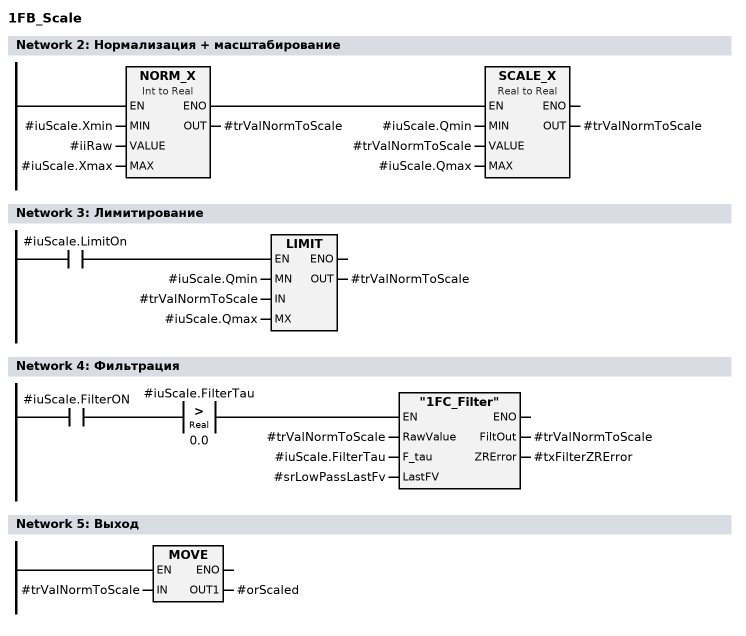
   RUNG wire#powerrail
      { S7_Templates := "[SrcType := Int, DestType := Real]" } Normalize(min := #iuScale.Xmin, value := #iiRaw, max := #iuScale.Xmax, out => #trValNormToScale)
      { S7_Templates := "[SrcType := Real, DestType := Real]" } Scale(min := #iuScale.Qmin, value := #trValNormToScale, max := #iuScale.Qmax, out => #trValNormToScale)
   END_RUNG
   // the same network as SCL:
   #trValNormToScale := NORM_X(MIN := #iuScale.Xmin, VALUE := #iiRaw, MAX := #iuScale.Xmax);
   #trValNormToScale := SCALE_X(MIN := #iuScale.Qmin, VALUE := #trValNormToScale, MAX := #iuScale.Qmax);
END_REGION

REGION Network 3: Лимитирование
   IF #iuScale.LimitOn THEN
       #trValNormToScale := LIMIT(MN := #iuScale.Qmin, IN := #trValNormToScale, MX := #iuScale.Qmax);
   END_IF;
END_REGION

REGION Network 4: Фильтрация
   RUNG wire#powerrail
      Contact( #iuScale.FilterON )
      { S7_Templates := "SrcType := Real" } GT_Contact(in1 := #iuScale.FilterTau, in2 := 0.0)
      "1FC_Filter"(RawValue := #trValNormToScale, F_tau := #iuScale.FilterTau, LastFV := #srLowPassLastFv, FiltOut => #trValNormToScale, ZRError => #txFilterZRError)
   END_RUNG
   // the same network as SCL:
   IF #iuScale.FilterON AND (#iuScale.FilterTau > 0.0) THEN
       "1FC_Filter"(RawValue := #trValNormToScale,
                    F_tau := #iuScale.FilterTau,
                    LastFV := #srLowPassLastFv,
                    FiltOut => #trValNormToScale,
                    ZRError => #txFilterZRError);
   END_IF;
END_REGION

REGION Network 5: Выход
   RUNG wire#powerrail
      Move(in := #trValNormToScale, out1 => #orScaled)
   END_RUNG
   // the same network as SCL:
   #orScaled := #trValNormToScale;
END_REGION
END_FUNCTION_BLOCK

FUNCTION_BLOCK "1FB_ScaleRTD"   // FB131, LAD
TITLE = Физ.значение аналогового входа термометра
{ S7_Optimized_Access := 'TRUE' }
VERSION : 0.1
// Преорбазование аналогового входа термрметра сопротивления в физ.значение согласно шкалы
   VAR_INPUT
      iiRaw : Int;   // Входной сигнал
      iuScale : "uScale";
   END_VAR
   VAR_OUTPUT
      orScaled : Real;   // Выходное отмасштабированное значение
   END_VAR
   VAR
      srLowPassLastFv : Real;   // Выходное значение для следующего цикла расчета
   END_VAR
   VAR_TEMP
      trValNormToScale : Real;   // Временная переменная
      txFilterZRError : Bool;   // Ошибка, если t = 0,0s
   END_VAR
BEGIN

REGION Network 2 (SCL): Временная переменная
   #trValNormToScale := INT_TO_REAL(#iiRaw);
END_REGION

REGION Network 3: Нормализация + масштабирование
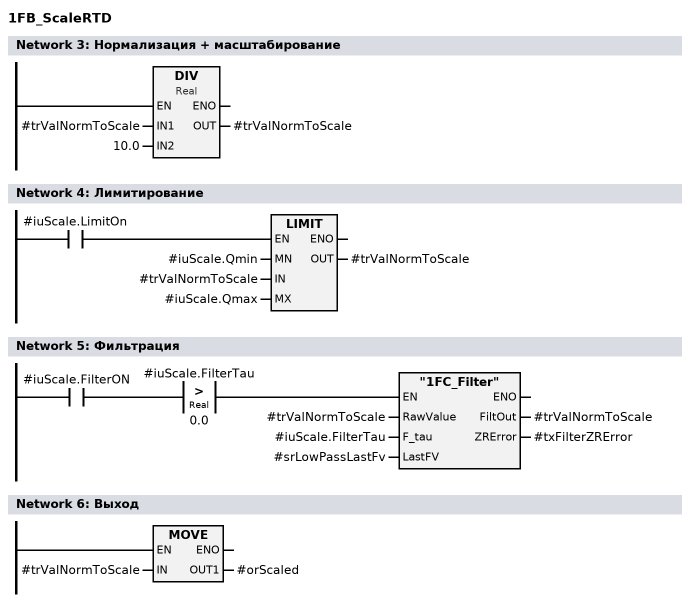
   RUNG wire#powerrail
      { S7_Templates := "SrcType := Real" } Div(in1 := #trValNormToScale, in2 := 10.0, out => #trValNormToScale)
   END_RUNG
   // the same network as SCL:
   #trValNormToScale := #trValNormToScale / 10.0;
END_REGION

REGION Network 4: Лимитирование
   IF #iuScale.LimitOn THEN
       #trValNormToScale := LIMIT(MN := #iuScale.Qmin, IN := #trValNormToScale, MX := #iuScale.Qmax);
   END_IF;
END_REGION

REGION Network 5: Фильтрация
   RUNG wire#powerrail
      Contact( #iuScale.FilterON )
      { S7_Templates := "SrcType := Real" } GT_Contact(in1 := #iuScale.FilterTau, in2 := 0.0)
      "1FC_Filter"(RawValue := #trValNormToScale, F_tau := #iuScale.FilterTau, LastFV := #srLowPassLastFv, FiltOut => #trValNormToScale, ZRError => #txFilterZRError)
   END_RUNG
   // the same network as SCL:
   IF #iuScale.FilterON AND (#iuScale.FilterTau > 0.0) THEN
       "1FC_Filter"(RawValue := #trValNormToScale,
                    F_tau := #iuScale.FilterTau,
                    LastFV := #srLowPassLastFv,
                    FiltOut => #trValNormToScale,
                    ZRError => #txFilterZRError);
   END_IF;
END_REGION

REGION Network 6: Выход
   RUNG wire#powerrail
      Move(in := #trValNormToScale, out1 => #orScaled)
   END_RUNG
   // the same network as SCL:
   #orScaled := #trValNormToScale;
END_REGION
END_FUNCTION_BLOCK

FUNCTION "1FC_Limit" : Void   // FC104, LAD
TITLE = Ааварийные и предупредительные границы
{ S7_Optimized_Access := 'TRUE' }
VERSION : 0.1
// Функция проверки аварийных и предупредительных границ аналогового сигнала, чтобы
// НШ <= НАГ <= НПГ <= ВПГ <= ВАГ <= КШ 
// НШ - начало шкалы
// НАГ - нижняя аварийная граница
// НПГ - нижняя предупредительная граница и тд
   VAR_INPUT
      inAI : "uScale";
   END_VAR
   VAR_IN_OUT
      ioWarning : "uWrnngAlarm";
      ioAlarm : "uWrnngAlarm";
   END_VAR
BEGIN

REGION Network 2: Если НАГ > НПГ и ниже если НАГ < НШ
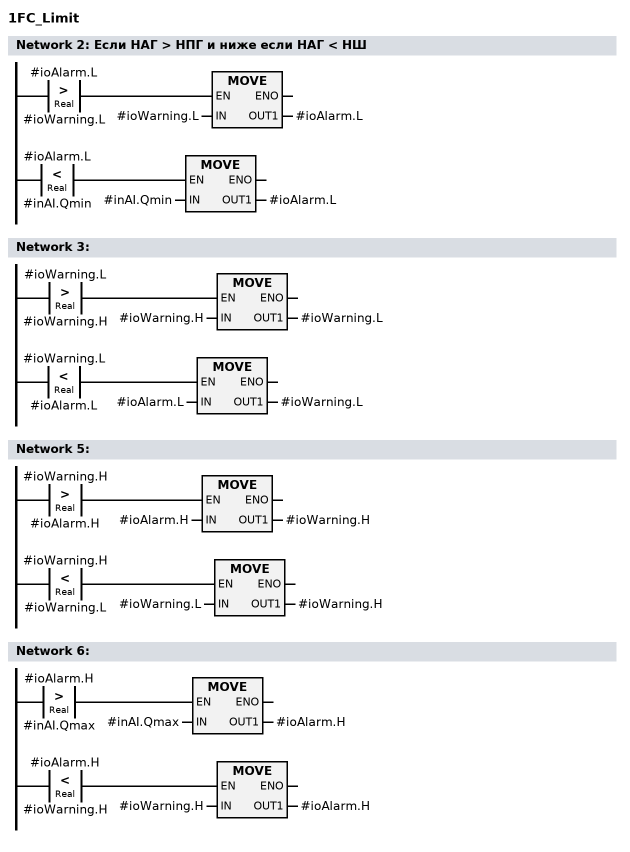
   RUNG wire#powerrail
      { S7_Templates := "SrcType := Real" } GT_Contact(in1 := #ioAlarm.L, in2 := #ioWarning.L)
      Move(in := #ioWarning.L, out1 => #ioAlarm.L)
   END_RUNG
   RUNG wire#powerrail
      { S7_Templates := "SrcType := Real" } LT_Contact(in1 := #ioAlarm.L, in2 := #inAI.Qmin)
      Move(in := #inAI.Qmin, out1 => #ioAlarm.L)
   END_RUNG
   // the same network as SCL:
   IF #ioAlarm.L > #ioWarning.L THEN #ioAlarm.L := #ioWarning.L; END_IF;
   IF #ioAlarm.L < #inAI.Qmin THEN #ioAlarm.L := #inAI.Qmin; END_IF;
END_REGION

REGION Network 3
   RUNG wire#powerrail
      { S7_Templates := "SrcType := Real" } GT_Contact(in1 := #ioWarning.L, in2 := #ioWarning.H)
      Move(in := #ioWarning.H, out1 => #ioWarning.L)
   END_RUNG
   RUNG wire#powerrail
      { S7_Templates := "SrcType := Real" } LT_Contact(in1 := #ioWarning.L, in2 := #ioAlarm.L)
      Move(in := #ioAlarm.L, out1 => #ioWarning.L)
   END_RUNG
   // the same network as SCL:
   IF #ioWarning.L > #ioWarning.H THEN #ioWarning.L := #ioWarning.H; END_IF;
   IF #ioWarning.L < #ioAlarm.L THEN #ioWarning.L := #ioAlarm.L; END_IF;
END_REGION

REGION Network 5
   RUNG wire#powerrail
      { S7_Templates := "SrcType := Real" } GT_Contact(in1 := #ioWarning.H, in2 := #ioAlarm.H)
      Move(in := #ioAlarm.H, out1 => #ioWarning.H)
   END_RUNG
   RUNG wire#powerrail
      { S7_Templates := "SrcType := Real" } LT_Contact(in1 := #ioWarning.H, in2 := #ioWarning.L)
      Move(in := #ioWarning.L, out1 => #ioWarning.H)
   END_RUNG
   // the same network as SCL:
   IF #ioWarning.H > #ioAlarm.H THEN #ioWarning.H := #ioAlarm.H; END_IF;
   IF #ioWarning.H < #ioWarning.L THEN #ioWarning.H := #ioWarning.L; END_IF;
END_REGION

REGION Network 6
   RUNG wire#powerrail
      { S7_Templates := "SrcType := Real" } GT_Contact(in1 := #ioAlarm.H, in2 := #inAI.Qmax)
      Move(in := #inAI.Qmax, out1 => #ioAlarm.H)
   END_RUNG
   RUNG wire#powerrail
      { S7_Templates := "SrcType := Real" } LT_Contact(in1 := #ioAlarm.H, in2 := #ioWarning.H)
      Move(in := #ioWarning.H, out1 => #ioAlarm.H)
   END_RUNG
   // the same network as SCL:
   IF #ioAlarm.H > #inAI.Qmax THEN #ioAlarm.H := #inAI.Qmax; END_IF;
   IF #ioAlarm.H < #ioWarning.H THEN #ioAlarm.H := #ioWarning.H; END_IF;
END_REGION
END_FUNCTION

FUNCTION "1FC_FlowNorm" : Void   // FC105, LAD
TITLE = Нормальный расход
{ S7_Optimized_Access := 'TRUE' }
VERSION : 0.1
// Нормализация расхода газа (не для расхода жидкости)
   VAR_INPUT
      inScaled : Real;
   END_VAR
   VAR_OUTPUT
      outScaledNorm : Real;
   END_VAR
BEGIN

REGION Network 2 (SCL)
   #outScaledNorm := #inScaled;
END_REGION
END_FUNCTION

FUNCTION "1FC_Filter" : Void   // FC106, SCL
TITLE = Фильтр низких частот
{ S7_Optimized_Access := 'TRUE' }
VERSION : 0.1
// Функция фильтрации аналогового входа
   VAR_INPUT
      RawValue : Real;   // Incoming unfiltered value
      F_tau : Real;   // Time interval (in seconds) for filter period
   END_VAR
   VAR_OUTPUT
      FiltOut : Real;   // Filtered output value
      ZRError : Bool;   // Error flag if F_tau is set to zero (invalid rate)
   END_VAR
   VAR_IN_OUT
      LastFV : Real;   // Static variable holds value of FiltOut from previous execution cycle.
   END_VAR
   VAR_TEMP
      ExpRate : Real;   // Equals exp(-0.1 / F_tau)
   END_VAR
BEGIN

   (* ============================================================================= *)
   (* PURPOSE : To filter a value by applying a first-order exponential filter      *)
   (*           with a user-selectable time period, F-tau. The filter is calculated *)
   (*           using the following formula -                                       *)
   (*                                                                               *)
   (*                                 Rate                    Rate                  *)
   (*           FiltOut := FiltOut * e     + RawValue * (1 - e     )                *)
   (*                                                                               *)
   (*           where Rate := (-0.1 / F_tau )                                       *)
   (*                                                                               *)
   (*           The Function Block is intended to be triggered every 100mS (hence   *)
   (*           the 0.1 in the formula) from cyclic interrupt Organization Block    *)
   (*           OB35. If a different resolution is required, use a different OB as  *)
   (*           the trigger, and adjust the formula to reflect this.                *)                                                                    
   (*                                                                               *)
   (* ============================================================================= *)


   IF #F_tau = 0.0 THEN                                        // If the filter period is set to zero ...
       #ZRError := true;                                     // .. . set the Zero Rate Error bit true
   ELSE
       #ZRError := false;                                       // Error bit reset to false
       #ExpRate := EXP(-0.1 / #F_tau);
       #FiltOut := #LastFV * #ExpRate + (#RawValue * (1 - #ExpRate)); // Calculate new output
       #LastFV := #FiltOut;                                       // Store output value for next cycle of calculation
   END_IF;
END_FUNCTION

FUNCTION "AI_Scaling" : Void   // FC131, LAD
TITLE = Физ.значение для всех аналог.сигналов
{ S7_Optimized_Access := 'TRUE' }
VERSION : 0.1
// Расчет физических значений всех аналоговых сигналов
   VAR_TEMP
      rTemp : Real;
   END_VAR
   VAR_TEMP   // added for the SCL form of the ladder/FBD networks
      _w1 : Bool;
   END_VAR
BEGIN

REGION Network 1: Разрежение на газоходе перед циклоном PIT201a
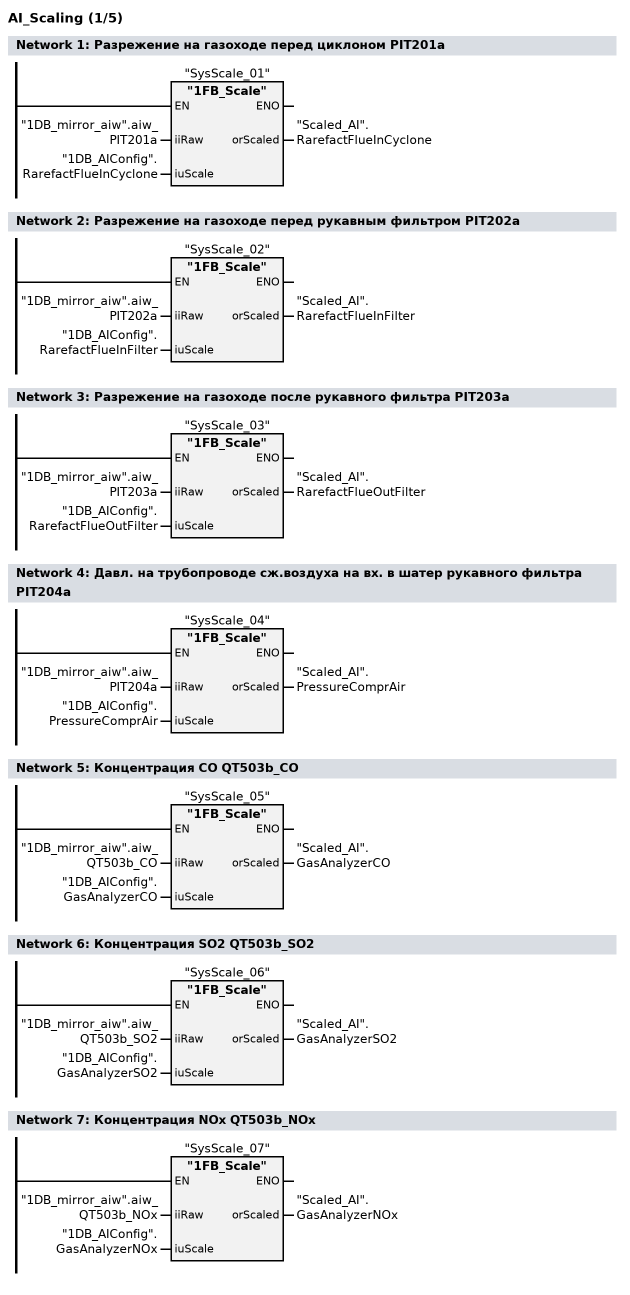
   RUNG wire#powerrail
      "SysScale_01"(iiRaw := "1DB_mirror_aiw".aiw_PIT201a, iuScale := "1DB_AIConfig".RarefactFlueInCyclone, orScaled => "Scaled_AI".RarefactFlueInCyclone)
   END_RUNG
   // the same network as SCL:
   "SysScale_01"(iiRaw := "1DB_mirror_aiw".aiw_PIT201a,   // "1FB_Scale"
                 iuScale := "1DB_AIConfig".RarefactFlueInCyclone,
                 orScaled => "Scaled_AI".RarefactFlueInCyclone);
END_REGION

REGION Network 2: Разрежение на газоходе перед рукавным фильтром PIT202a
   RUNG wire#powerrail
      "SysScale_02"(iiRaw := "1DB_mirror_aiw".aiw_PIT202a, iuScale := "1DB_AIConfig".RarefactFlueInFilter, orScaled => "Scaled_AI".RarefactFlueInFilter)
   END_RUNG
   // the same network as SCL:
   "SysScale_02"(iiRaw := "1DB_mirror_aiw".aiw_PIT202a,   // "1FB_Scale"
                 iuScale := "1DB_AIConfig".RarefactFlueInFilter,
                 orScaled => "Scaled_AI".RarefactFlueInFilter);
END_REGION

REGION Network 3: Разрежение на газоходе после рукавного фильтра PIT203a
   RUNG wire#powerrail
      "SysScale_03"(iiRaw := "1DB_mirror_aiw".aiw_PIT203a, iuScale := "1DB_AIConfig".RarefactFlueOutFilter, orScaled => "Scaled_AI".RarefactFlueOutFilter)
   END_RUNG
   // the same network as SCL:
   "SysScale_03"(iiRaw := "1DB_mirror_aiw".aiw_PIT203a,   // "1FB_Scale"
                 iuScale := "1DB_AIConfig".RarefactFlueOutFilter,
                 orScaled => "Scaled_AI".RarefactFlueOutFilter);
END_REGION

REGION Network 4: Давл. на трубопроводе сж.воздуха на вх. в шатер рукавного фильтра PIT204a
   RUNG wire#powerrail
      "SysScale_04"(iiRaw := "1DB_mirror_aiw".aiw_PIT204a, iuScale := "1DB_AIConfig".PressureComprAir, orScaled => "Scaled_AI".PressureComprAir)
   END_RUNG
   // the same network as SCL:
   "SysScale_04"(iiRaw := "1DB_mirror_aiw".aiw_PIT204a,   // "1FB_Scale"
                 iuScale := "1DB_AIConfig".PressureComprAir,
                 orScaled => "Scaled_AI".PressureComprAir);
END_REGION

REGION Network 5: Концентрация CO QT503b_CO
   RUNG wire#powerrail
      "SysScale_05"(iiRaw := "1DB_mirror_aiw".aiw_QT503b_CO, iuScale := "1DB_AIConfig".GasAnalyzerCO, orScaled => "Scaled_AI".GasAnalyzerCO)
   END_RUNG
   // the same network as SCL:
   "SysScale_05"(iiRaw := "1DB_mirror_aiw".aiw_QT503b_CO,   // "1FB_Scale"
                 iuScale := "1DB_AIConfig".GasAnalyzerCO,
                 orScaled => "Scaled_AI".GasAnalyzerCO);
END_REGION

REGION Network 6: Концентрация SO2 QT503b_SO2
   RUNG wire#powerrail
      "SysScale_06"(iiRaw := "1DB_mirror_aiw".aiw_QT503b_SO2, iuScale := "1DB_AIConfig".GasAnalyzerSO2, orScaled => "Scaled_AI".GasAnalyzerSO2)
   END_RUNG
   // the same network as SCL:
   "SysScale_06"(iiRaw := "1DB_mirror_aiw".aiw_QT503b_SO2,   // "1FB_Scale"
                 iuScale := "1DB_AIConfig".GasAnalyzerSO2,
                 orScaled => "Scaled_AI".GasAnalyzerSO2);
END_REGION

REGION Network 7: Концентрация NOx QT503b_NOx
   RUNG wire#powerrail
      "SysScale_07"(iiRaw := "1DB_mirror_aiw".aiw_QT503b_NOx, iuScale := "1DB_AIConfig".GasAnalyzerNOx, orScaled => "Scaled_AI".GasAnalyzerNOx)
   END_RUNG
   // the same network as SCL:
   "SysScale_07"(iiRaw := "1DB_mirror_aiw".aiw_QT503b_NOx,   // "1FB_Scale"
                 iuScale := "1DB_AIConfig".GasAnalyzerNOx,
                 orScaled => "Scaled_AI".GasAnalyzerNOx);
END_REGION

REGION Network 8: Концентрация CO2 QT503b_CO2
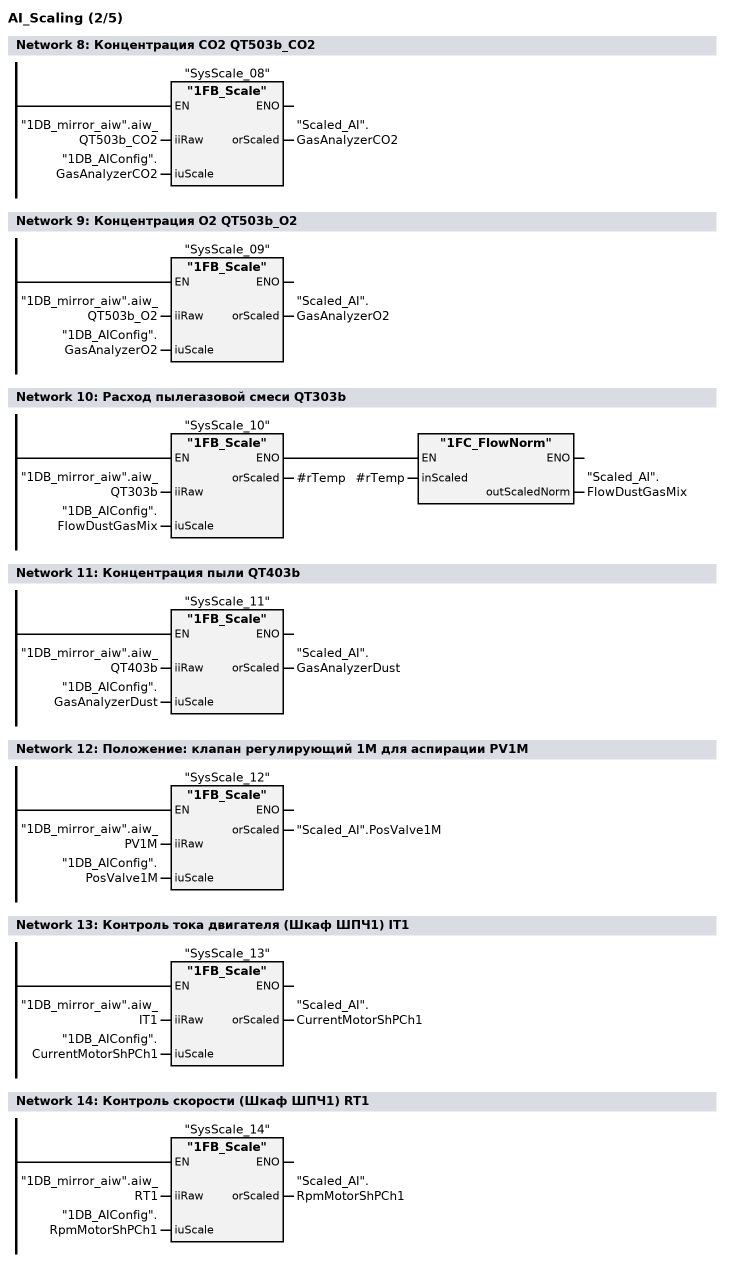
   RUNG wire#powerrail
      "SysScale_08"(iiRaw := "1DB_mirror_aiw".aiw_QT503b_CO2, iuScale := "1DB_AIConfig".GasAnalyzerCO2, orScaled => "Scaled_AI".GasAnalyzerCO2)
   END_RUNG
   // the same network as SCL:
   "SysScale_08"(iiRaw := "1DB_mirror_aiw".aiw_QT503b_CO2,   // "1FB_Scale"
                 iuScale := "1DB_AIConfig".GasAnalyzerCO2,
                 orScaled => "Scaled_AI".GasAnalyzerCO2);
END_REGION

REGION Network 9: Концентрация O2 QT503b_O2
   RUNG wire#powerrail
      "SysScale_09"(iiRaw := "1DB_mirror_aiw".aiw_QT503b_O2, iuScale := "1DB_AIConfig".GasAnalyzerO2, orScaled => "Scaled_AI".GasAnalyzerO2)
   END_RUNG
   // the same network as SCL:
   "SysScale_09"(iiRaw := "1DB_mirror_aiw".aiw_QT503b_O2,   // "1FB_Scale"
                 iuScale := "1DB_AIConfig".GasAnalyzerO2,
                 orScaled => "Scaled_AI".GasAnalyzerO2);
END_REGION

REGION Network 10: Расход пылегазовой смеси QT303b
   RUNG wire#powerrail
      "SysScale_10"(iiRaw := "1DB_mirror_aiw".aiw_QT303b, iuScale := "1DB_AIConfig".FlowDustGasMix, orScaled => #rTemp)
      "1FC_FlowNorm"(inScaled := #rTemp, outScaledNorm => "Scaled_AI".FlowDustGasMix)
   END_RUNG
   // the same network as SCL:
   "SysScale_10"(iiRaw := "1DB_mirror_aiw".aiw_QT303b,   // "1FB_Scale"
                 iuScale := "1DB_AIConfig".FlowDustGasMix,
                 orScaled => #rTemp,
                 ENO => #_w1);
   IF #_w1 THEN "1FC_FlowNorm"(inScaled := #rTemp, outScaledNorm => "Scaled_AI".FlowDustGasMix); END_IF;
END_REGION

REGION Network 11: Концентрация пыли QT403b
   RUNG wire#powerrail
      "SysScale_11"(iiRaw := "1DB_mirror_aiw".aiw_QT403b, iuScale := "1DB_AIConfig".GasAnalyzerDust, orScaled => "Scaled_AI".GasAnalyzerDust)
   END_RUNG
   // the same network as SCL:
   "SysScale_11"(iiRaw := "1DB_mirror_aiw".aiw_QT403b,   // "1FB_Scale"
                 iuScale := "1DB_AIConfig".GasAnalyzerDust,
                 orScaled => "Scaled_AI".GasAnalyzerDust);
END_REGION

REGION Network 12: Положение: клапан регулирующий 1M для аспирации PV1M
   RUNG wire#powerrail
      "SysScale_12"(iiRaw := "1DB_mirror_aiw".aiw_PV1M, iuScale := "1DB_AIConfig".PosValve1M, orScaled => "Scaled_AI".PosValve1M)
   END_RUNG
   // the same network as SCL:
   "SysScale_12"(iiRaw := "1DB_mirror_aiw".aiw_PV1M,   // "1FB_Scale"
                 iuScale := "1DB_AIConfig".PosValve1M,
                 orScaled => "Scaled_AI".PosValve1M);
END_REGION

REGION Network 13: Контроль тока двигателя (Шкаф ШПЧ1) IT1
   RUNG wire#powerrail
      "SysScale_13"(iiRaw := "1DB_mirror_aiw".aiw_IT1, iuScale := "1DB_AIConfig".CurrentMotorShPCh1, orScaled => "Scaled_AI".CurrentMotorShPCh1)
   END_RUNG
   // the same network as SCL:
   "SysScale_13"(iiRaw := "1DB_mirror_aiw".aiw_IT1,   // "1FB_Scale"
                 iuScale := "1DB_AIConfig".CurrentMotorShPCh1,
                 orScaled => "Scaled_AI".CurrentMotorShPCh1);
END_REGION

REGION Network 14: Контроль скорости (Шкаф ШПЧ1) RT1
   RUNG wire#powerrail
      "SysScale_14"(iiRaw := "1DB_mirror_aiw".aiw_RT1, iuScale := "1DB_AIConfig".RpmMotorShPCh1, orScaled => "Scaled_AI".RpmMotorShPCh1)
   END_RUNG
   // the same network as SCL:
   "SysScale_14"(iiRaw := "1DB_mirror_aiw".aiw_RT1,   // "1FB_Scale"
                 iuScale := "1DB_AIConfig".RpmMotorShPCh1,
                 orScaled => "Scaled_AI".RpmMotorShPCh1);
END_REGION

REGION Network 15: 2 резервных места
END_REGION

REGION Network 16: 2 резервных места
END_REGION

REGION Network 17: Дымосос 1. Вибрация переднего подшипника вентилятора X-направления VE801a
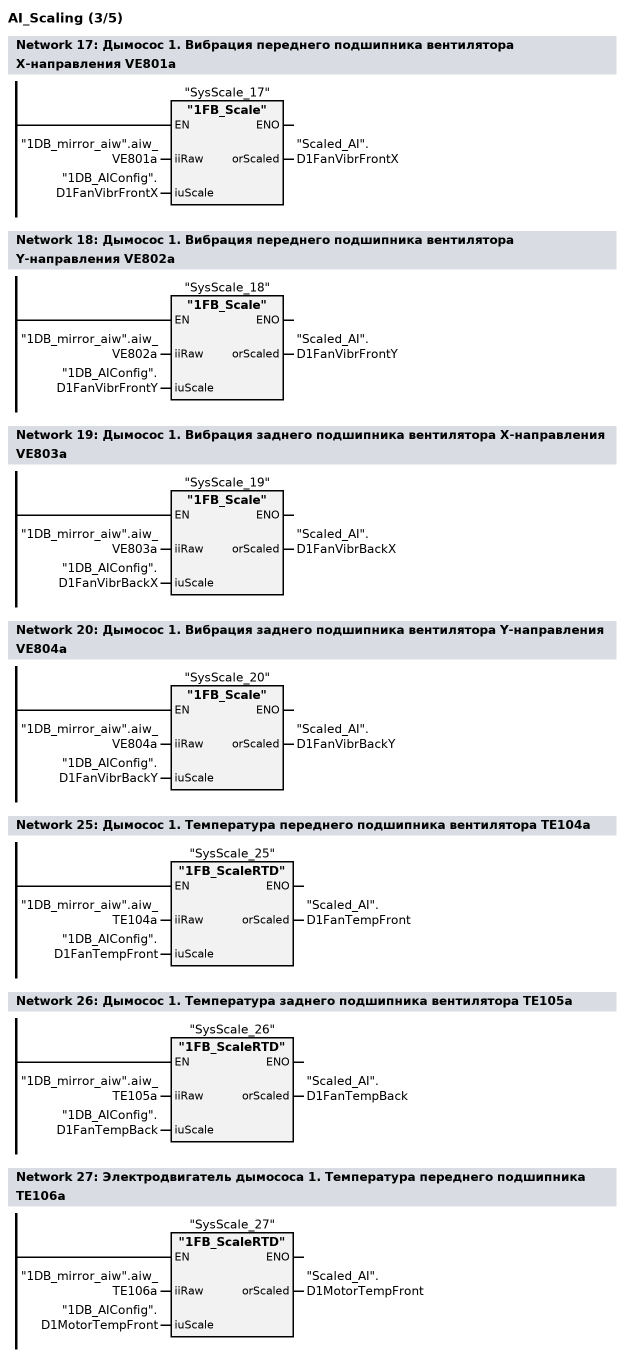
   RUNG wire#powerrail
      "SysScale_17"(iiRaw := "1DB_mirror_aiw".aiw_VE801a, iuScale := "1DB_AIConfig".D1FanVibrFrontX, orScaled => "Scaled_AI".D1FanVibrFrontX)
   END_RUNG
   // the same network as SCL:
   "SysScale_17"(iiRaw := "1DB_mirror_aiw".aiw_VE801a,   // "1FB_Scale"
                 iuScale := "1DB_AIConfig".D1FanVibrFrontX,
                 orScaled => "Scaled_AI".D1FanVibrFrontX);
END_REGION

REGION Network 18: Дымосос 1. Вибрация переднего подшипника вентилятора Y-направления VE802a
   RUNG wire#powerrail
      "SysScale_18"(iiRaw := "1DB_mirror_aiw".aiw_VE802a, iuScale := "1DB_AIConfig".D1FanVibrFrontY, orScaled => "Scaled_AI".D1FanVibrFrontY)
   END_RUNG
   // the same network as SCL:
   "SysScale_18"(iiRaw := "1DB_mirror_aiw".aiw_VE802a,   // "1FB_Scale"
                 iuScale := "1DB_AIConfig".D1FanVibrFrontY,
                 orScaled => "Scaled_AI".D1FanVibrFrontY);
END_REGION

REGION Network 19: Дымосос 1. Вибрация заднего подшипника вентилятора X-направления VE803a
   RUNG wire#powerrail
      "SysScale_19"(iiRaw := "1DB_mirror_aiw".aiw_VE803a, iuScale := "1DB_AIConfig".D1FanVibrBackX, orScaled => "Scaled_AI".D1FanVibrBackX)
   END_RUNG
   // the same network as SCL:
   "SysScale_19"(iiRaw := "1DB_mirror_aiw".aiw_VE803a,   // "1FB_Scale"
                 iuScale := "1DB_AIConfig".D1FanVibrBackX,
                 orScaled => "Scaled_AI".D1FanVibrBackX);
END_REGION

REGION Network 20: Дымосос 1. Вибрация заднего подшипника вентилятора Y-направления VE804a
   RUNG wire#powerrail
      "SysScale_20"(iiRaw := "1DB_mirror_aiw".aiw_VE804a, iuScale := "1DB_AIConfig".D1FanVibrBackY, orScaled => "Scaled_AI".D1FanVibrBackY)
   END_RUNG
   // the same network as SCL:
   "SysScale_20"(iiRaw := "1DB_mirror_aiw".aiw_VE804a,   // "1FB_Scale"
                 iuScale := "1DB_AIConfig".D1FanVibrBackY,
                 orScaled => "Scaled_AI".D1FanVibrBackY);
END_REGION

REGION Network 21: 4 резервных места
END_REGION

REGION Network 22: 4 резервных места
END_REGION

REGION Network 23: 4 резервных места
END_REGION

REGION Network 24: 4 резервных места
END_REGION

REGION Network 25: Дымосос 1. Температура переднего подшипника вентилятора TE104a
   RUNG wire#powerrail
      "SysScale_25"(iiRaw := "1DB_mirror_aiw".aiw_TE104a, iuScale := "1DB_AIConfig".D1FanTempFront, orScaled => "Scaled_AI".D1FanTempFront)
   END_RUNG
   // the same network as SCL:
   "SysScale_25"(iiRaw := "1DB_mirror_aiw".aiw_TE104a,   // "1FB_ScaleRTD"
                 iuScale := "1DB_AIConfig".D1FanTempFront,
                 orScaled => "Scaled_AI".D1FanTempFront);
END_REGION

REGION Network 26: Дымосос 1. Температура заднего подшипника вентилятора TE105a
   RUNG wire#powerrail
      "SysScale_26"(iiRaw := "1DB_mirror_aiw".aiw_TE105a, iuScale := "1DB_AIConfig".D1FanTempBack, orScaled => "Scaled_AI".D1FanTempBack)
   END_RUNG
   // the same network as SCL:
   "SysScale_26"(iiRaw := "1DB_mirror_aiw".aiw_TE105a,   // "1FB_ScaleRTD"
                 iuScale := "1DB_AIConfig".D1FanTempBack,
                 orScaled => "Scaled_AI".D1FanTempBack);
END_REGION

REGION Network 27: Электродвигатель дымососа 1. Температура переднего подшипника TE106a
   RUNG wire#powerrail
      "SysScale_27"(iiRaw := "1DB_mirror_aiw".aiw_TE106a, iuScale := "1DB_AIConfig".D1MotorTempFront, orScaled => "Scaled_AI".D1MotorTempFront)
   END_RUNG
   // the same network as SCL:
   "SysScale_27"(iiRaw := "1DB_mirror_aiw".aiw_TE106a,   // "1FB_ScaleRTD"
                 iuScale := "1DB_AIConfig".D1MotorTempFront,
                 orScaled => "Scaled_AI".D1MotorTempFront);
END_REGION

REGION Network 28: Электродвигатель дымососа 1. Температура заднего подшипника TE107a
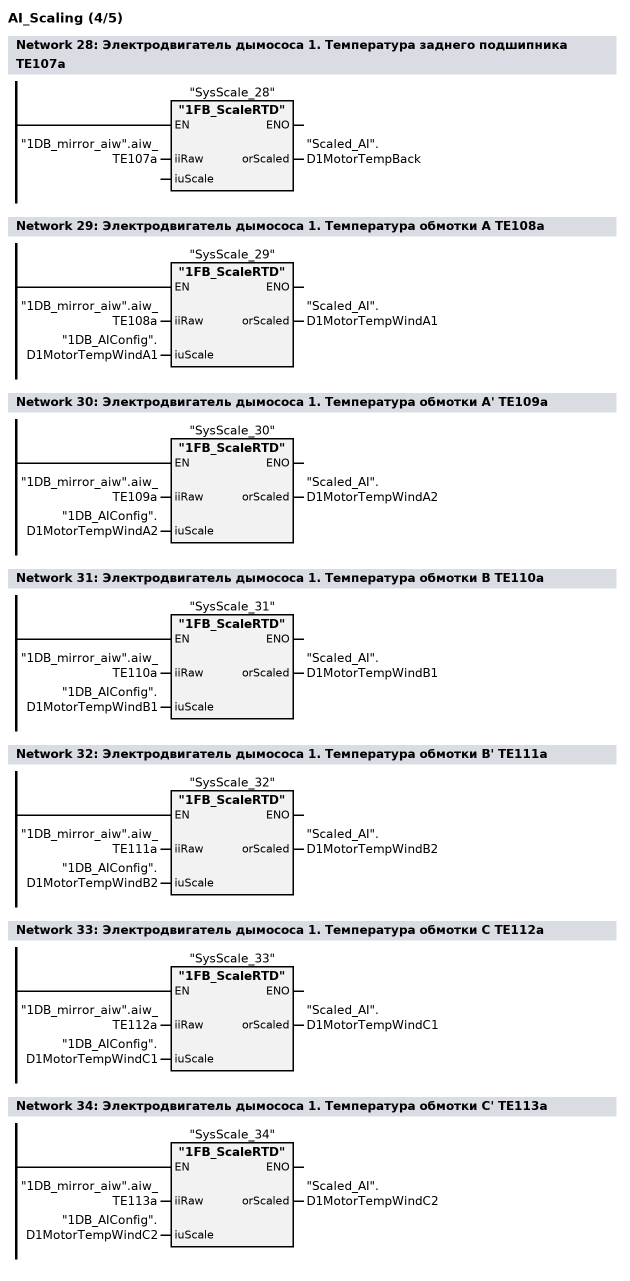
   RUNG wire#powerrail
      "SysScale_28"(iiRaw := "1DB_mirror_aiw".aiw_TE107a, iuScale :=, orScaled => "Scaled_AI".D1MotorTempBack)
   END_RUNG
   // the same network as SCL:
   "SysScale_28"(iiRaw := "1DB_mirror_aiw".aiw_TE107a, orScaled => "Scaled_AI".D1MotorTempBack);   // "1FB_ScaleRTD"
END_REGION

REGION Network 29: Электродвигатель дымососа 1. Температура обмотки А TE108a
   RUNG wire#powerrail
      "SysScale_29"(iiRaw := "1DB_mirror_aiw".aiw_TE108a, iuScale := "1DB_AIConfig".D1MotorTempWindA1, orScaled => "Scaled_AI".D1MotorTempWindA1)
   END_RUNG
   // the same network as SCL:
   "SysScale_29"(iiRaw := "1DB_mirror_aiw".aiw_TE108a,   // "1FB_ScaleRTD"
                 iuScale := "1DB_AIConfig".D1MotorTempWindA1,
                 orScaled => "Scaled_AI".D1MotorTempWindA1);
END_REGION

REGION Network 30: Электродвигатель дымососа 1. Температура обмотки А' TE109a
   RUNG wire#powerrail
      "SysScale_30"(iiRaw := "1DB_mirror_aiw".aiw_TE109a, iuScale := "1DB_AIConfig".D1MotorTempWindA2, orScaled => "Scaled_AI".D1MotorTempWindA2)
   END_RUNG
   // the same network as SCL:
   "SysScale_30"(iiRaw := "1DB_mirror_aiw".aiw_TE109a,   // "1FB_ScaleRTD"
                 iuScale := "1DB_AIConfig".D1MotorTempWindA2,
                 orScaled => "Scaled_AI".D1MotorTempWindA2);
END_REGION

REGION Network 31: Электродвигатель дымососа 1. Температура обмотки B TE110a
   RUNG wire#powerrail
      "SysScale_31"(iiRaw := "1DB_mirror_aiw".aiw_TE110a, iuScale := "1DB_AIConfig".D1MotorTempWindB1, orScaled => "Scaled_AI".D1MotorTempWindB1)
   END_RUNG
   // the same network as SCL:
   "SysScale_31"(iiRaw := "1DB_mirror_aiw".aiw_TE110a,   // "1FB_ScaleRTD"
                 iuScale := "1DB_AIConfig".D1MotorTempWindB1,
                 orScaled => "Scaled_AI".D1MotorTempWindB1);
END_REGION

REGION Network 32: Электродвигатель дымососа 1. Температура обмотки B' TE111a
   RUNG wire#powerrail
      "SysScale_32"(iiRaw := "1DB_mirror_aiw".aiw_TE111a, iuScale := "1DB_AIConfig".D1MotorTempWindB2, orScaled => "Scaled_AI".D1MotorTempWindB2)
   END_RUNG
   // the same network as SCL:
   "SysScale_32"(iiRaw := "1DB_mirror_aiw".aiw_TE111a,   // "1FB_ScaleRTD"
                 iuScale := "1DB_AIConfig".D1MotorTempWindB2,
                 orScaled => "Scaled_AI".D1MotorTempWindB2);
END_REGION

REGION Network 33: Электродвигатель дымососа 1. Температура обмотки C TE112a
   RUNG wire#powerrail
      "SysScale_33"(iiRaw := "1DB_mirror_aiw".aiw_TE112a, iuScale := "1DB_AIConfig".D1MotorTempWindC1, orScaled => "Scaled_AI".D1MotorTempWindC1)
   END_RUNG
   // the same network as SCL:
   "SysScale_33"(iiRaw := "1DB_mirror_aiw".aiw_TE112a,   // "1FB_ScaleRTD"
                 iuScale := "1DB_AIConfig".D1MotorTempWindC1,
                 orScaled => "Scaled_AI".D1MotorTempWindC1);
END_REGION

REGION Network 34: Электродвигатель дымососа 1. Температура обмотки C' TE113a
   RUNG wire#powerrail
      "SysScale_34"(iiRaw := "1DB_mirror_aiw".aiw_TE113a, iuScale := "1DB_AIConfig".D1MotorTempWindC2, orScaled => "Scaled_AI".D1MotorTempWindC2)
   END_RUNG
   // the same network as SCL:
   "SysScale_34"(iiRaw := "1DB_mirror_aiw".aiw_TE113a,   // "1FB_ScaleRTD"
                 iuScale := "1DB_AIConfig".D1MotorTempWindC2,
                 orScaled => "Scaled_AI".D1MotorTempWindC2);
END_REGION

REGION Network 35: 2 резервных места
END_REGION

REGION Network 36: 2 резервных места
END_REGION

REGION Network 37: Температура на газоходе перед циклоном TE101a
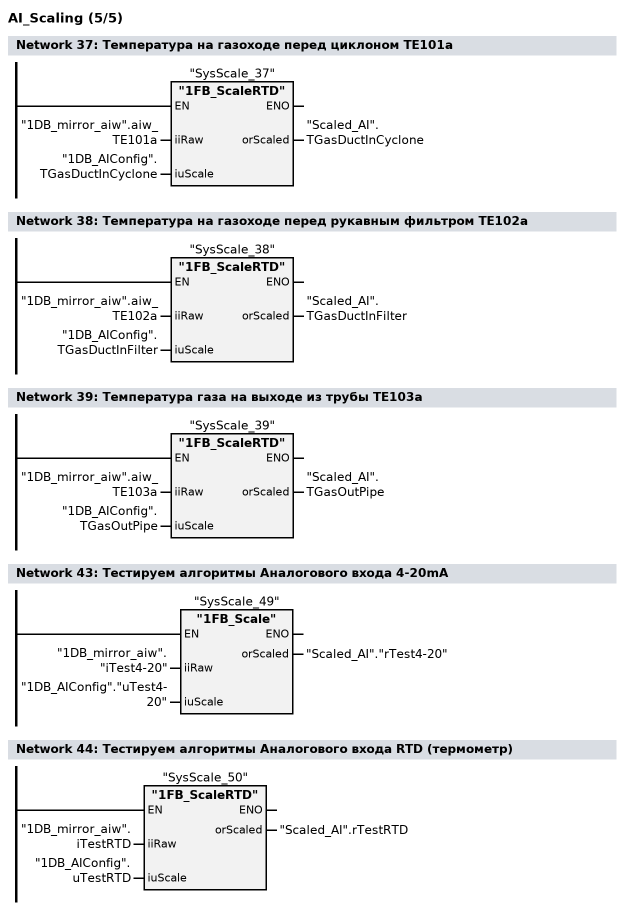
   RUNG wire#powerrail
      "SysScale_37"(iiRaw := "1DB_mirror_aiw".aiw_TE101a, iuScale := "1DB_AIConfig".TGasDuctInCyclone, orScaled => "Scaled_AI".TGasDuctInCyclone)
   END_RUNG
   // the same network as SCL:
   "SysScale_37"(iiRaw := "1DB_mirror_aiw".aiw_TE101a,   // "1FB_ScaleRTD"
                 iuScale := "1DB_AIConfig".TGasDuctInCyclone,
                 orScaled => "Scaled_AI".TGasDuctInCyclone);
END_REGION

REGION Network 38: Температура на газоходе перед рукавным фильтром TE102a
   RUNG wire#powerrail
      "SysScale_38"(iiRaw := "1DB_mirror_aiw".aiw_TE102a, iuScale := "1DB_AIConfig".TGasDuctInFilter, orScaled => "Scaled_AI".TGasDuctInFilter)
   END_RUNG
   // the same network as SCL:
   "SysScale_38"(iiRaw := "1DB_mirror_aiw".aiw_TE102a,   // "1FB_ScaleRTD"
                 iuScale := "1DB_AIConfig".TGasDuctInFilter,
                 orScaled => "Scaled_AI".TGasDuctInFilter);
END_REGION

REGION Network 39: Температура газа на выходе из трубы TE103a
   RUNG wire#powerrail
      "SysScale_39"(iiRaw := "1DB_mirror_aiw".aiw_TE103a, iuScale := "1DB_AIConfig".TGasOutPipe, orScaled => "Scaled_AI".TGasOutPipe)
   END_RUNG
   // the same network as SCL:
   "SysScale_39"(iiRaw := "1DB_mirror_aiw".aiw_TE103a,   // "1FB_ScaleRTD"
                 iuScale := "1DB_AIConfig".TGasOutPipe,
                 orScaled => "Scaled_AI".TGasOutPipe);
END_REGION

REGION Network 43: Тестируем алгоритмы Аналогового входа 4-20mA
   RUNG wire#powerrail
      "SysScale_49"(iiRaw := "1DB_mirror_aiw"."iTest4-20", iuScale := "1DB_AIConfig"."uTest4-20", orScaled => "Scaled_AI"."rTest4-20")
   END_RUNG
   // the same network as SCL:
   "SysScale_49"(iiRaw := "1DB_mirror_aiw"."iTest4-20",   // "1FB_Scale"
                 iuScale := "1DB_AIConfig"."uTest4-20",
                 orScaled => "Scaled_AI"."rTest4-20");
END_REGION

REGION Network 44: Тестируем алгоритмы Аналогового входа RTD (термометр)
   RUNG wire#powerrail
      "SysScale_50"(iiRaw := "1DB_mirror_aiw".iTestRTD, iuScale := "1DB_AIConfig".uTestRTD, orScaled => "Scaled_AI".rTestRTD)
   END_RUNG
   // the same network as SCL:
   "SysScale_50"(iiRaw := "1DB_mirror_aiw".iTestRTD,   // "1FB_ScaleRTD"
                 iuScale := "1DB_AIConfig".uTestRTD,
                 orScaled => "Scaled_AI".rTestRTD);
END_REGION
END_FUNCTION

FUNCTION "AI_Limiting" : Void   // FC132, LAD
TITLE = Аварийные и предупр.границы всех аналоговых сигналов
{ S7_Optimized_Access := 'TRUE' }
VERSION : 0.1
// Проверка аварийных и предупредительных границ для всех аналоговых сигналов
BEGIN

REGION Network 2: Разрежение на газоходе перед циклоном PIT201a
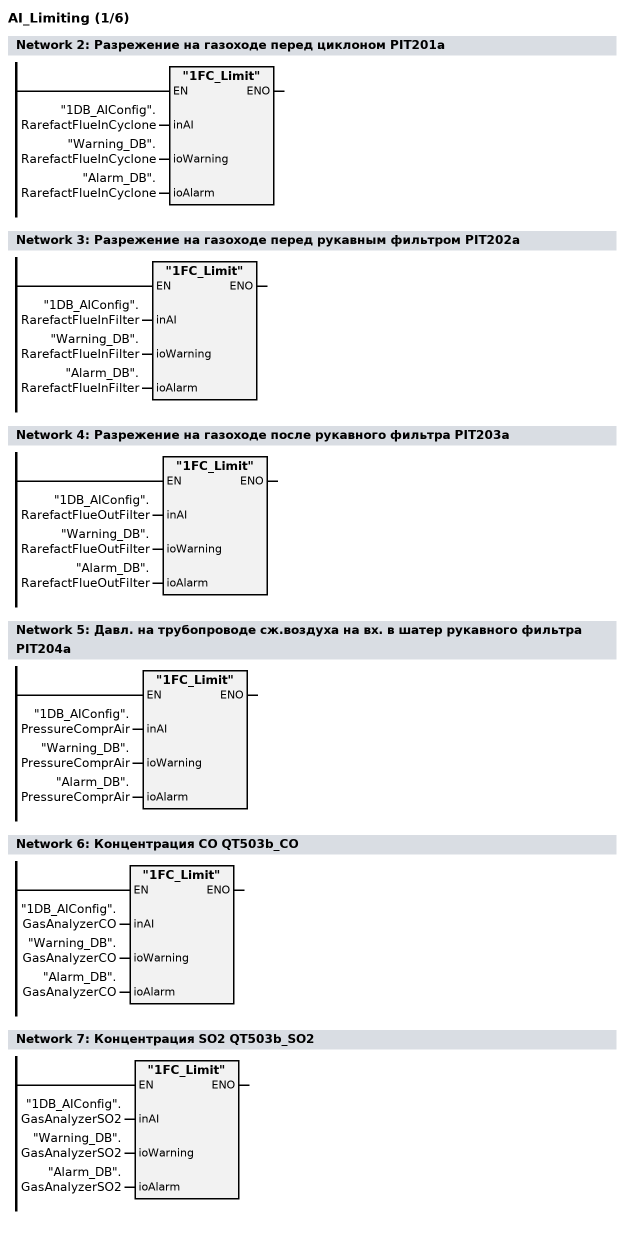
   RUNG wire#powerrail
      "1FC_Limit"(inAI := "1DB_AIConfig".RarefactFlueInCyclone, ioWarning := "Warning_DB".RarefactFlueInCyclone, ioAlarm := "Alarm_DB".RarefactFlueInCyclone)
   END_RUNG
   // the same network as SCL:
   "1FC_Limit"(inAI := "1DB_AIConfig".RarefactFlueInCyclone,
               ioWarning := "Warning_DB".RarefactFlueInCyclone,
               ioAlarm := "Alarm_DB".RarefactFlueInCyclone);
END_REGION

REGION Network 3: Разрежение на газоходе перед рукавным фильтром PIT202a
   RUNG wire#powerrail
      "1FC_Limit"(inAI := "1DB_AIConfig".RarefactFlueInFilter, ioWarning := "Warning_DB".RarefactFlueInFilter, ioAlarm := "Alarm_DB".RarefactFlueInFilter)
   END_RUNG
   // the same network as SCL:
   "1FC_Limit"(inAI := "1DB_AIConfig".RarefactFlueInFilter,
               ioWarning := "Warning_DB".RarefactFlueInFilter,
               ioAlarm := "Alarm_DB".RarefactFlueInFilter);
END_REGION

REGION Network 4: Разрежение на газоходе после рукавного фильтра PIT203a
   RUNG wire#powerrail
      "1FC_Limit"(inAI := "1DB_AIConfig".RarefactFlueOutFilter, ioWarning := "Warning_DB".RarefactFlueOutFilter, ioAlarm := "Alarm_DB".RarefactFlueOutFilter)
   END_RUNG
   // the same network as SCL:
   "1FC_Limit"(inAI := "1DB_AIConfig".RarefactFlueOutFilter,
               ioWarning := "Warning_DB".RarefactFlueOutFilter,
               ioAlarm := "Alarm_DB".RarefactFlueOutFilter);
END_REGION

REGION Network 5: Давл. на трубопроводе сж.воздуха на вх. в шатер рукавного фильтра PIT204a
   RUNG wire#powerrail
      "1FC_Limit"(inAI := "1DB_AIConfig".PressureComprAir, ioWarning := "Warning_DB".PressureComprAir, ioAlarm := "Alarm_DB".PressureComprAir)
   END_RUNG
   // the same network as SCL:
   "1FC_Limit"(inAI := "1DB_AIConfig".PressureComprAir,
               ioWarning := "Warning_DB".PressureComprAir,
               ioAlarm := "Alarm_DB".PressureComprAir);
END_REGION

REGION Network 6: Концентрация CO QT503b_CO
   RUNG wire#powerrail
      "1FC_Limit"(inAI := "1DB_AIConfig".GasAnalyzerCO, ioWarning := "Warning_DB".GasAnalyzerCO, ioAlarm := "Alarm_DB".GasAnalyzerCO)
   END_RUNG
   // the same network as SCL:
   "1FC_Limit"(inAI := "1DB_AIConfig".GasAnalyzerCO,
               ioWarning := "Warning_DB".GasAnalyzerCO,
               ioAlarm := "Alarm_DB".GasAnalyzerCO);
END_REGION

REGION Network 7: Концентрация SO2 QT503b_SO2
   RUNG wire#powerrail
      "1FC_Limit"(inAI := "1DB_AIConfig".GasAnalyzerSO2, ioWarning := "Warning_DB".GasAnalyzerSO2, ioAlarm := "Alarm_DB".GasAnalyzerSO2)
   END_RUNG
   // the same network as SCL:
   "1FC_Limit"(inAI := "1DB_AIConfig".GasAnalyzerSO2,
               ioWarning := "Warning_DB".GasAnalyzerSO2,
               ioAlarm := "Alarm_DB".GasAnalyzerSO2);
END_REGION

REGION Network 8: Концентрация NOx QT503b_NOx
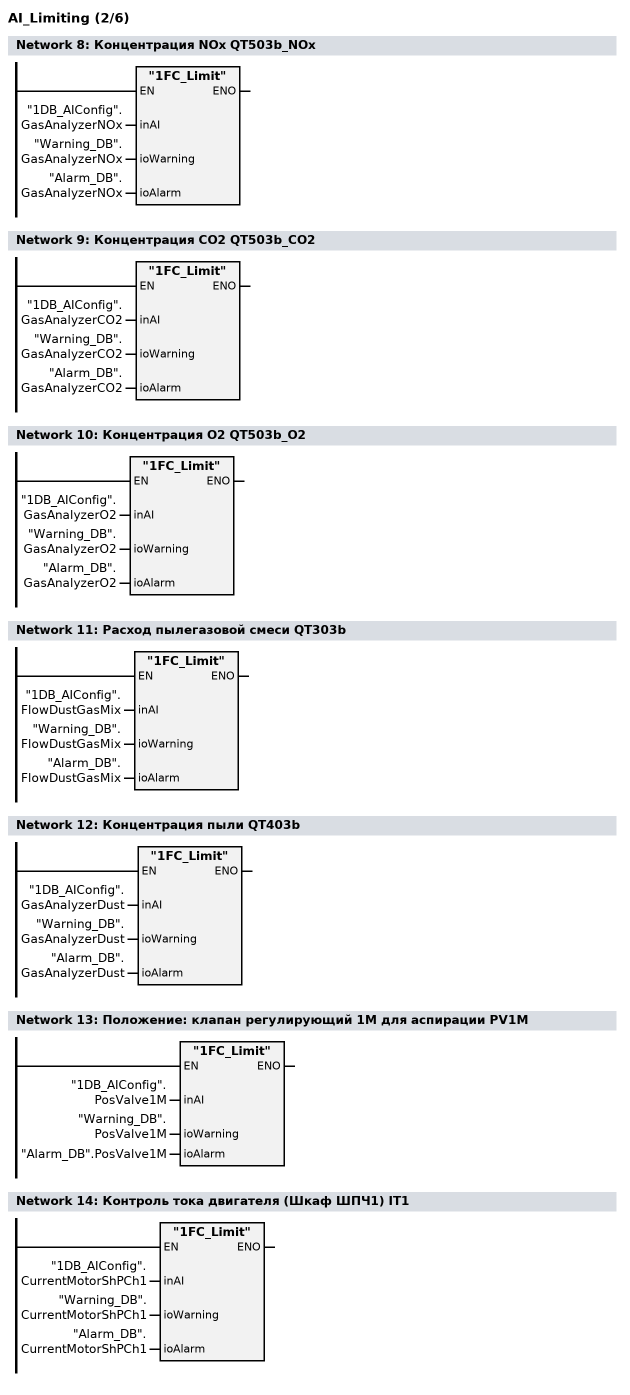
   RUNG wire#powerrail
      "1FC_Limit"(inAI := "1DB_AIConfig".GasAnalyzerNOx, ioWarning := "Warning_DB".GasAnalyzerNOx, ioAlarm := "Alarm_DB".GasAnalyzerNOx)
   END_RUNG
   // the same network as SCL:
   "1FC_Limit"(inAI := "1DB_AIConfig".GasAnalyzerNOx,
               ioWarning := "Warning_DB".GasAnalyzerNOx,
               ioAlarm := "Alarm_DB".GasAnalyzerNOx);
END_REGION

REGION Network 9: Концентрация CO2 QT503b_CO2
   RUNG wire#powerrail
      "1FC_Limit"(inAI := "1DB_AIConfig".GasAnalyzerCO2, ioWarning := "Warning_DB".GasAnalyzerCO2, ioAlarm := "Alarm_DB".GasAnalyzerCO2)
   END_RUNG
   // the same network as SCL:
   "1FC_Limit"(inAI := "1DB_AIConfig".GasAnalyzerCO2,
               ioWarning := "Warning_DB".GasAnalyzerCO2,
               ioAlarm := "Alarm_DB".GasAnalyzerCO2);
END_REGION

REGION Network 10: Концентрация O2 QT503b_O2
   RUNG wire#powerrail
      "1FC_Limit"(inAI := "1DB_AIConfig".GasAnalyzerO2, ioWarning := "Warning_DB".GasAnalyzerO2, ioAlarm := "Alarm_DB".GasAnalyzerO2)
   END_RUNG
   // the same network as SCL:
   "1FC_Limit"(inAI := "1DB_AIConfig".GasAnalyzerO2,
               ioWarning := "Warning_DB".GasAnalyzerO2,
               ioAlarm := "Alarm_DB".GasAnalyzerO2);
END_REGION

REGION Network 11: Расход пылегазовой смеси QT303b
   RUNG wire#powerrail
      "1FC_Limit"(inAI := "1DB_AIConfig".FlowDustGasMix, ioWarning := "Warning_DB".FlowDustGasMix, ioAlarm := "Alarm_DB".FlowDustGasMix)
   END_RUNG
   // the same network as SCL:
   "1FC_Limit"(inAI := "1DB_AIConfig".FlowDustGasMix,
               ioWarning := "Warning_DB".FlowDustGasMix,
               ioAlarm := "Alarm_DB".FlowDustGasMix);
END_REGION

REGION Network 12: Концентрация пыли QT403b
   RUNG wire#powerrail
      "1FC_Limit"(inAI := "1DB_AIConfig".GasAnalyzerDust, ioWarning := "Warning_DB".GasAnalyzerDust, ioAlarm := "Alarm_DB".GasAnalyzerDust)
   END_RUNG
   // the same network as SCL:
   "1FC_Limit"(inAI := "1DB_AIConfig".GasAnalyzerDust,
               ioWarning := "Warning_DB".GasAnalyzerDust,
               ioAlarm := "Alarm_DB".GasAnalyzerDust);
END_REGION

REGION Network 13: Положение: клапан регулирующий 1M для аспирации PV1M
   RUNG wire#powerrail
      "1FC_Limit"(inAI := "1DB_AIConfig".PosValve1M, ioWarning := "Warning_DB".PosValve1M, ioAlarm := "Alarm_DB".PosValve1M)
   END_RUNG
   // the same network as SCL:
   "1FC_Limit"(inAI := "1DB_AIConfig".PosValve1M,
               ioWarning := "Warning_DB".PosValve1M,
               ioAlarm := "Alarm_DB".PosValve1M);
END_REGION

REGION Network 14: Контроль тока двигателя (Шкаф ШПЧ1) IT1
   RUNG wire#powerrail
      "1FC_Limit"(inAI := "1DB_AIConfig".CurrentMotorShPCh1, ioWarning := "Warning_DB".CurrentMotorShPCh1, ioAlarm := "Alarm_DB".CurrentMotorShPCh1)
   END_RUNG
   // the same network as SCL:
   "1FC_Limit"(inAI := "1DB_AIConfig".CurrentMotorShPCh1,
               ioWarning := "Warning_DB".CurrentMotorShPCh1,
               ioAlarm := "Alarm_DB".CurrentMotorShPCh1);
END_REGION

REGION Network 15: Контроль скорости (Шкаф ШПЧ1) RT1
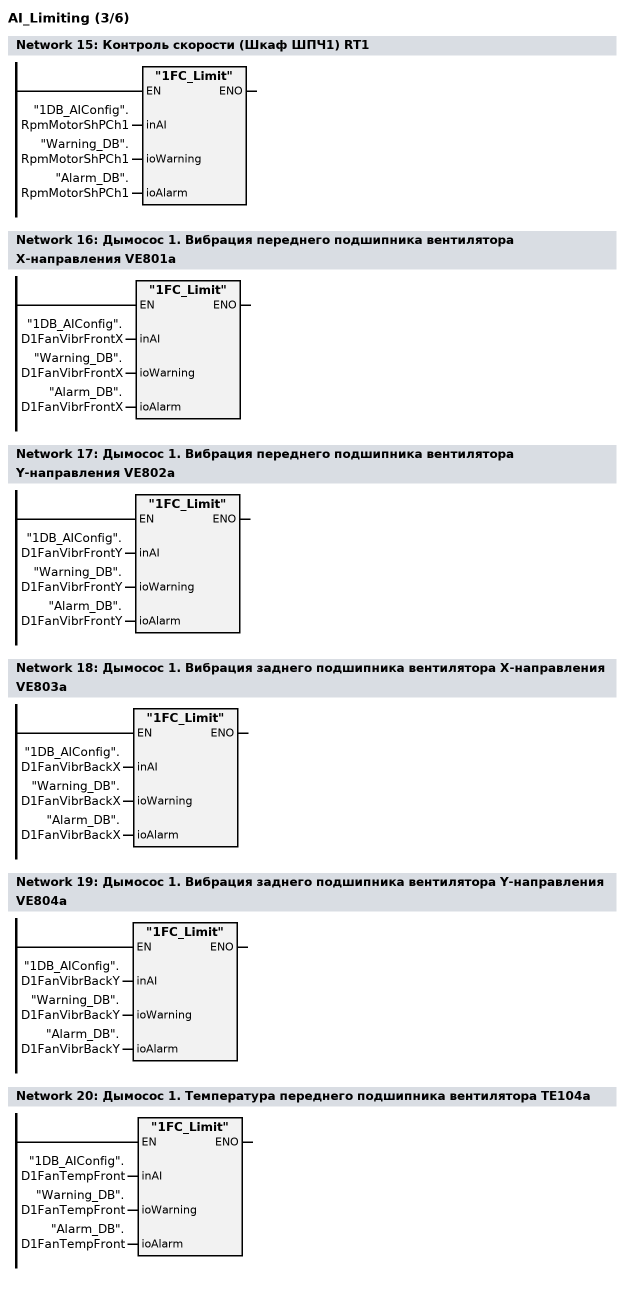
   RUNG wire#powerrail
      "1FC_Limit"(inAI := "1DB_AIConfig".RpmMotorShPCh1, ioWarning := "Warning_DB".RpmMotorShPCh1, ioAlarm := "Alarm_DB".RpmMotorShPCh1)
   END_RUNG
   // the same network as SCL:
   "1FC_Limit"(inAI := "1DB_AIConfig".RpmMotorShPCh1,
               ioWarning := "Warning_DB".RpmMotorShPCh1,
               ioAlarm := "Alarm_DB".RpmMotorShPCh1);
END_REGION

REGION Network 16: Дымосос 1. Вибрация переднего подшипника вентилятора X-направления VE801a
   RUNG wire#powerrail
      "1FC_Limit"(inAI := "1DB_AIConfig".D1FanVibrFrontX, ioWarning := "Warning_DB".D1FanVibrFrontX, ioAlarm := "Alarm_DB".D1FanVibrFrontX)
   END_RUNG
   // the same network as SCL:
   "1FC_Limit"(inAI := "1DB_AIConfig".D1FanVibrFrontX,
               ioWarning := "Warning_DB".D1FanVibrFrontX,
               ioAlarm := "Alarm_DB".D1FanVibrFrontX);
END_REGION

REGION Network 17: Дымосос 1. Вибрация переднего подшипника вентилятора Y-направления VE802a
   RUNG wire#powerrail
      "1FC_Limit"(inAI := "1DB_AIConfig".D1FanVibrFrontY, ioWarning := "Warning_DB".D1FanVibrFrontY, ioAlarm := "Alarm_DB".D1FanVibrFrontY)
   END_RUNG
   // the same network as SCL:
   "1FC_Limit"(inAI := "1DB_AIConfig".D1FanVibrFrontY,
               ioWarning := "Warning_DB".D1FanVibrFrontY,
               ioAlarm := "Alarm_DB".D1FanVibrFrontY);
END_REGION

REGION Network 18: Дымосос 1. Вибрация заднего подшипника вентилятора X-направления VE803a
   RUNG wire#powerrail
      "1FC_Limit"(inAI := "1DB_AIConfig".D1FanVibrBackX, ioWarning := "Warning_DB".D1FanVibrBackX, ioAlarm := "Alarm_DB".D1FanVibrBackX)
   END_RUNG
   // the same network as SCL:
   "1FC_Limit"(inAI := "1DB_AIConfig".D1FanVibrBackX,
               ioWarning := "Warning_DB".D1FanVibrBackX,
               ioAlarm := "Alarm_DB".D1FanVibrBackX);
END_REGION

REGION Network 19: Дымосос 1. Вибрация заднего подшипника вентилятора Y-направления VE804a
   RUNG wire#powerrail
      "1FC_Limit"(inAI := "1DB_AIConfig".D1FanVibrBackY, ioWarning := "Warning_DB".D1FanVibrBackY, ioAlarm := "Alarm_DB".D1FanVibrBackY)
   END_RUNG
   // the same network as SCL:
   "1FC_Limit"(inAI := "1DB_AIConfig".D1FanVibrBackY,
               ioWarning := "Warning_DB".D1FanVibrBackY,
               ioAlarm := "Alarm_DB".D1FanVibrBackY);
END_REGION

REGION Network 20: Дымосос 1. Температура переднего подшипника вентилятора TE104a
   RUNG wire#powerrail
      "1FC_Limit"(inAI := "1DB_AIConfig".D1FanTempFront, ioWarning := "Warning_DB".D1FanTempFront, ioAlarm := "Alarm_DB".D1FanTempFront)
   END_RUNG
   // the same network as SCL:
   "1FC_Limit"(inAI := "1DB_AIConfig".D1FanTempFront,
               ioWarning := "Warning_DB".D1FanTempFront,
               ioAlarm := "Alarm_DB".D1FanTempFront);
END_REGION

REGION Network 21: Дымосос 1. Температура заднего подшипника вентилятора TE105a
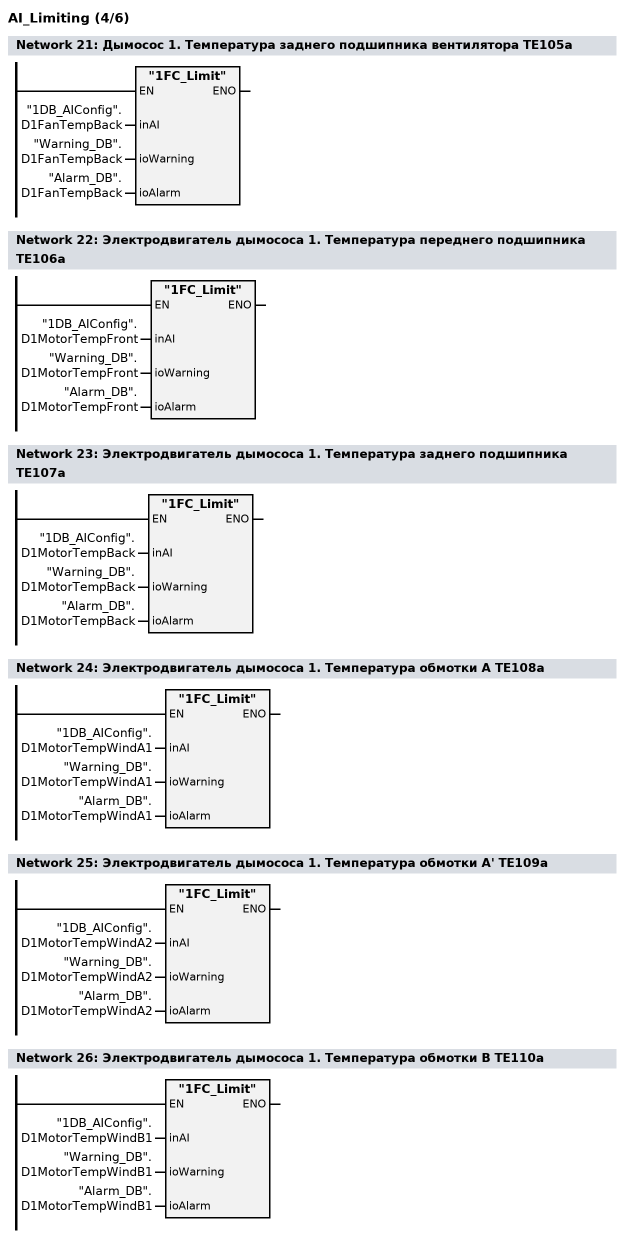
   RUNG wire#powerrail
      "1FC_Limit"(inAI := "1DB_AIConfig".D1FanTempBack, ioWarning := "Warning_DB".D1FanTempBack, ioAlarm := "Alarm_DB".D1FanTempBack)
   END_RUNG
   // the same network as SCL:
   "1FC_Limit"(inAI := "1DB_AIConfig".D1FanTempBack,
               ioWarning := "Warning_DB".D1FanTempBack,
               ioAlarm := "Alarm_DB".D1FanTempBack);
END_REGION

REGION Network 22: Электродвигатель дымососа 1. Температура переднего подшипника TE106a
   RUNG wire#powerrail
      "1FC_Limit"(inAI := "1DB_AIConfig".D1MotorTempFront, ioWarning := "Warning_DB".D1MotorTempFront, ioAlarm := "Alarm_DB".D1MotorTempFront)
   END_RUNG
   // the same network as SCL:
   "1FC_Limit"(inAI := "1DB_AIConfig".D1MotorTempFront,
               ioWarning := "Warning_DB".D1MotorTempFront,
               ioAlarm := "Alarm_DB".D1MotorTempFront);
END_REGION

REGION Network 23: Электродвигатель дымососа 1. Температура заднего подшипника TE107a
   RUNG wire#powerrail
      "1FC_Limit"(inAI := "1DB_AIConfig".D1MotorTempBack, ioWarning := "Warning_DB".D1MotorTempBack, ioAlarm := "Alarm_DB".D1MotorTempBack)
   END_RUNG
   // the same network as SCL:
   "1FC_Limit"(inAI := "1DB_AIConfig".D1MotorTempBack,
               ioWarning := "Warning_DB".D1MotorTempBack,
               ioAlarm := "Alarm_DB".D1MotorTempBack);
END_REGION

REGION Network 24: Электродвигатель дымососа 1. Температура обмотки А TE108a
   RUNG wire#powerrail
      "1FC_Limit"(inAI := "1DB_AIConfig".D1MotorTempWindA1, ioWarning := "Warning_DB".D1MotorTempWindA1, ioAlarm := "Alarm_DB".D1MotorTempWindA1)
   END_RUNG
   // the same network as SCL:
   "1FC_Limit"(inAI := "1DB_AIConfig".D1MotorTempWindA1,
               ioWarning := "Warning_DB".D1MotorTempWindA1,
               ioAlarm := "Alarm_DB".D1MotorTempWindA1);
END_REGION

REGION Network 25: Электродвигатель дымососа 1. Температура обмотки А' TE109a
   RUNG wire#powerrail
      "1FC_Limit"(inAI := "1DB_AIConfig".D1MotorTempWindA2, ioWarning := "Warning_DB".D1MotorTempWindA2, ioAlarm := "Alarm_DB".D1MotorTempWindA2)
   END_RUNG
   // the same network as SCL:
   "1FC_Limit"(inAI := "1DB_AIConfig".D1MotorTempWindA2,
               ioWarning := "Warning_DB".D1MotorTempWindA2,
               ioAlarm := "Alarm_DB".D1MotorTempWindA2);
END_REGION

REGION Network 26: Электродвигатель дымососа 1. Температура обмотки B TE110a
   RUNG wire#powerrail
      "1FC_Limit"(inAI := "1DB_AIConfig".D1MotorTempWindB1, ioWarning := "Warning_DB".D1MotorTempWindB1, ioAlarm := "Alarm_DB".D1MotorTempWindB1)
   END_RUNG
   // the same network as SCL:
   "1FC_Limit"(inAI := "1DB_AIConfig".D1MotorTempWindB1,
               ioWarning := "Warning_DB".D1MotorTempWindB1,
               ioAlarm := "Alarm_DB".D1MotorTempWindB1);
END_REGION

REGION Network 27: Электродвигатель дымососа 1. Температура обмотки B' TE111a
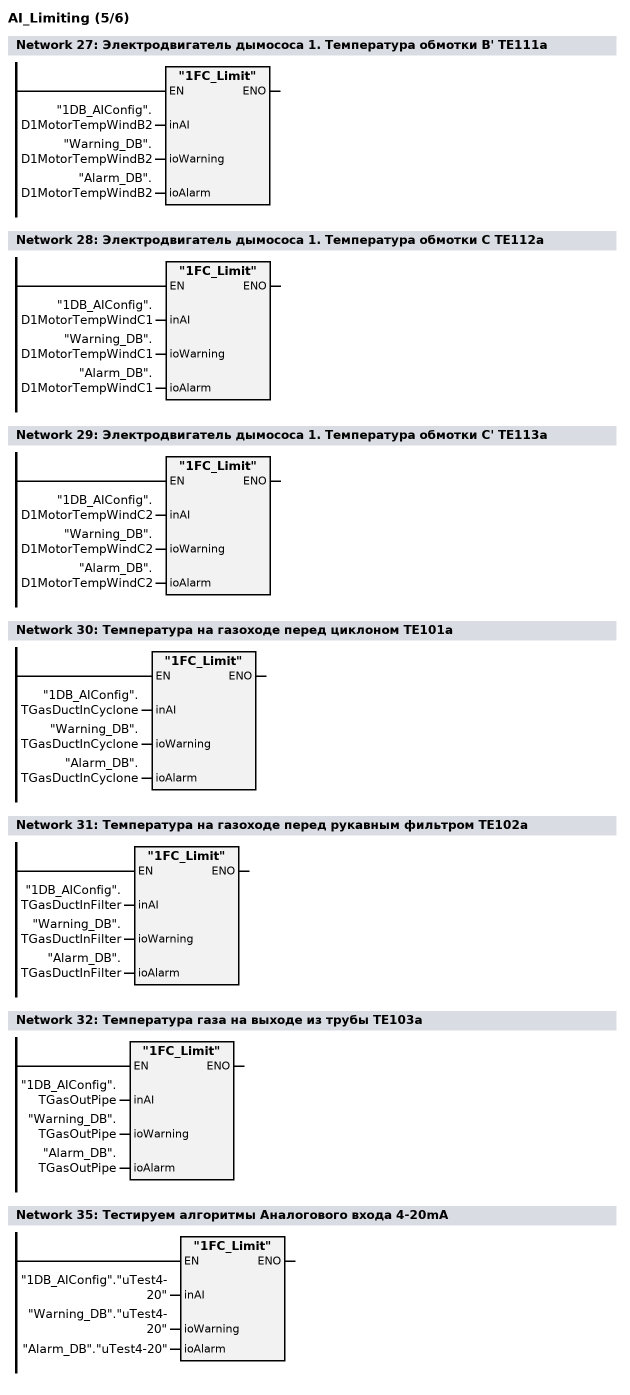
   RUNG wire#powerrail
      "1FC_Limit"(inAI := "1DB_AIConfig".D1MotorTempWindB2, ioWarning := "Warning_DB".D1MotorTempWindB2, ioAlarm := "Alarm_DB".D1MotorTempWindB2)
   END_RUNG
   // the same network as SCL:
   "1FC_Limit"(inAI := "1DB_AIConfig".D1MotorTempWindB2,
               ioWarning := "Warning_DB".D1MotorTempWindB2,
               ioAlarm := "Alarm_DB".D1MotorTempWindB2);
END_REGION

REGION Network 28: Электродвигатель дымососа 1. Температура обмотки C TE112a
   RUNG wire#powerrail
      "1FC_Limit"(inAI := "1DB_AIConfig".D1MotorTempWindC1, ioWarning := "Warning_DB".D1MotorTempWindC1, ioAlarm := "Alarm_DB".D1MotorTempWindC1)
   END_RUNG
   // the same network as SCL:
   "1FC_Limit"(inAI := "1DB_AIConfig".D1MotorTempWindC1,
               ioWarning := "Warning_DB".D1MotorTempWindC1,
               ioAlarm := "Alarm_DB".D1MotorTempWindC1);
END_REGION

REGION Network 29: Электродвигатель дымососа 1. Температура обмотки C' TE113a
   RUNG wire#powerrail
      "1FC_Limit"(inAI := "1DB_AIConfig".D1MotorTempWindC2, ioWarning := "Warning_DB".D1MotorTempWindC2, ioAlarm := "Alarm_DB".D1MotorTempWindC2)
   END_RUNG
   // the same network as SCL:
   "1FC_Limit"(inAI := "1DB_AIConfig".D1MotorTempWindC2,
               ioWarning := "Warning_DB".D1MotorTempWindC2,
               ioAlarm := "Alarm_DB".D1MotorTempWindC2);
END_REGION

REGION Network 30: Температура на газоходе перед циклоном TE101a
   RUNG wire#powerrail
      "1FC_Limit"(inAI := "1DB_AIConfig".TGasDuctInCyclone, ioWarning := "Warning_DB".TGasDuctInCyclone, ioAlarm := "Alarm_DB".TGasDuctInCyclone)
   END_RUNG
   // the same network as SCL:
   "1FC_Limit"(inAI := "1DB_AIConfig".TGasDuctInCyclone,
               ioWarning := "Warning_DB".TGasDuctInCyclone,
               ioAlarm := "Alarm_DB".TGasDuctInCyclone);
END_REGION

REGION Network 31: Температура на газоходе перед рукавным фильтром TE102a
   RUNG wire#powerrail
      "1FC_Limit"(inAI := "1DB_AIConfig".TGasDuctInFilter, ioWarning := "Warning_DB".TGasDuctInFilter, ioAlarm := "Alarm_DB".TGasDuctInFilter)
   END_RUNG
   // the same network as SCL:
   "1FC_Limit"(inAI := "1DB_AIConfig".TGasDuctInFilter,
               ioWarning := "Warning_DB".TGasDuctInFilter,
               ioAlarm := "Alarm_DB".TGasDuctInFilter);
END_REGION

REGION Network 32: Температура газа на выходе из трубы TE103a
   RUNG wire#powerrail
      "1FC_Limit"(inAI := "1DB_AIConfig".TGasOutPipe, ioWarning := "Warning_DB".TGasOutPipe, ioAlarm := "Alarm_DB".TGasOutPipe)
   END_RUNG
   // the same network as SCL:
   "1FC_Limit"(inAI := "1DB_AIConfig".TGasOutPipe,
               ioWarning := "Warning_DB".TGasOutPipe,
               ioAlarm := "Alarm_DB".TGasOutPipe);
END_REGION

REGION Network 35: Тестируем алгоритмы Аналогового входа 4-20mA
   RUNG wire#powerrail
      "1FC_Limit"(inAI := "1DB_AIConfig"."uTest4-20", ioWarning := "Warning_DB"."uTest4-20", ioAlarm := "Alarm_DB"."uTest4-20")
   END_RUNG
   // the same network as SCL:
   "1FC_Limit"(inAI := "1DB_AIConfig"."uTest4-20",
               ioWarning := "Warning_DB"."uTest4-20",
               ioAlarm := "Alarm_DB"."uTest4-20");
END_REGION

REGION Network 36: Тестируем алгоритмы Аналогового входа RTD (термометр)
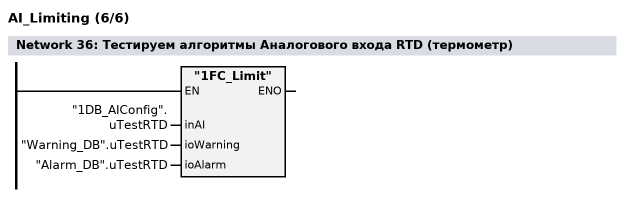
   RUNG wire#powerrail
      "1FC_Limit"(inAI := "1DB_AIConfig".uTestRTD, ioWarning := "Warning_DB".uTestRTD, ioAlarm := "Alarm_DB".uTestRTD)
   END_RUNG
   // the same network as SCL:
   "1FC_Limit"(inAI := "1DB_AIConfig".uTestRTD,
               ioWarning := "Warning_DB".uTestRTD,
               ioAlarm := "Alarm_DB".uTestRTD);
END_REGION
END_FUNCTION

FUNCTION "AI_Controling" : Void   // FC133, LAD
TITLE = Авар.и предупр.границы для всех аналог.сигналов
{ S7_Optimized_Access := 'TRUE' }
VERSION : 0.1
// Прверка всех аналоговых сигналов на аврийные и предупредительные границы
BEGIN

REGION Network 1: Разрежение на газоходе перед циклоном PIT201a
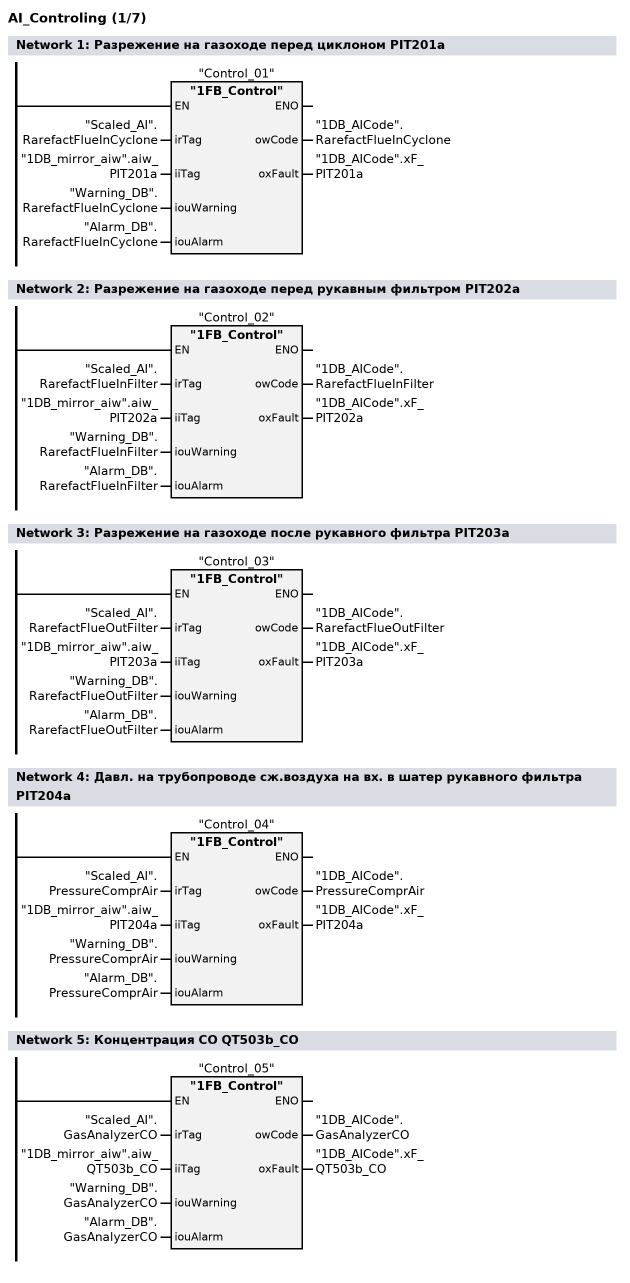
   RUNG wire#powerrail
      "Control_01"(irTag := "Scaled_AI".RarefactFlueInCyclone, iiTag := "1DB_mirror_aiw".aiw_PIT201a, iouWarning := "Warning_DB".RarefactFlueInCyclone, iouAlarm := "Alarm_DB".RarefactFlueInCyclone, owCode => "1DB_AICode".RarefactFlueInCyclone, oxFault => "1DB_AICode".xF_PIT201a)
   END_RUNG
   // the same network as SCL:
   "Control_01"(irTag := "Scaled_AI".RarefactFlueInCyclone,   // "1FB_Control"
                iiTag := "1DB_mirror_aiw".aiw_PIT201a,
                iouWarning := "Warning_DB".RarefactFlueInCyclone,
                iouAlarm := "Alarm_DB".RarefactFlueInCyclone,
                owCode => "1DB_AICode".RarefactFlueInCyclone,
                oxFault => "1DB_AICode".xF_PIT201a);
END_REGION

REGION Network 2: Разрежение на газоходе перед рукавным фильтром PIT202a
   RUNG wire#powerrail
      "Control_02"(irTag := "Scaled_AI".RarefactFlueInFilter, iiTag := "1DB_mirror_aiw".aiw_PIT202a, iouWarning := "Warning_DB".RarefactFlueInFilter, iouAlarm := "Alarm_DB".RarefactFlueInFilter, owCode => "1DB_AICode".RarefactFlueInFilter, oxFault => "1DB_AICode".xF_PIT202a)
   END_RUNG
   // the same network as SCL:
   "Control_02"(irTag := "Scaled_AI".RarefactFlueInFilter,   // "1FB_Control"
                iiTag := "1DB_mirror_aiw".aiw_PIT202a,
                iouWarning := "Warning_DB".RarefactFlueInFilter,
                iouAlarm := "Alarm_DB".RarefactFlueInFilter,
                owCode => "1DB_AICode".RarefactFlueInFilter,
                oxFault => "1DB_AICode".xF_PIT202a);
END_REGION

REGION Network 3: Разрежение на газоходе после рукавного фильтра PIT203a
   RUNG wire#powerrail
      "Control_03"(irTag := "Scaled_AI".RarefactFlueOutFilter, iiTag := "1DB_mirror_aiw".aiw_PIT203a, iouWarning := "Warning_DB".RarefactFlueOutFilter, iouAlarm := "Alarm_DB".RarefactFlueOutFilter, owCode => "1DB_AICode".RarefactFlueOutFilter, oxFault => "1DB_AICode".xF_PIT203a)
   END_RUNG
   // the same network as SCL:
   "Control_03"(irTag := "Scaled_AI".RarefactFlueOutFilter,   // "1FB_Control"
                iiTag := "1DB_mirror_aiw".aiw_PIT203a,
                iouWarning := "Warning_DB".RarefactFlueOutFilter,
                iouAlarm := "Alarm_DB".RarefactFlueOutFilter,
                owCode => "1DB_AICode".RarefactFlueOutFilter,
                oxFault => "1DB_AICode".xF_PIT203a);
END_REGION

REGION Network 4: Давл. на трубопроводе сж.воздуха на вх. в шатер рукавного фильтра PIT204a
   RUNG wire#powerrail
      "Control_04"(irTag := "Scaled_AI".PressureComprAir, iiTag := "1DB_mirror_aiw".aiw_PIT204a, iouWarning := "Warning_DB".PressureComprAir, iouAlarm := "Alarm_DB".PressureComprAir, owCode => "1DB_AICode".PressureComprAir, oxFault => "1DB_AICode".xF_PIT204a)
   END_RUNG
   // the same network as SCL:
   "Control_04"(irTag := "Scaled_AI".PressureComprAir,   // "1FB_Control"
                iiTag := "1DB_mirror_aiw".aiw_PIT204a,
                iouWarning := "Warning_DB".PressureComprAir,
                iouAlarm := "Alarm_DB".PressureComprAir,
                owCode => "1DB_AICode".PressureComprAir,
                oxFault => "1DB_AICode".xF_PIT204a);
END_REGION

REGION Network 5: Концентрация CO QT503b_CO
   RUNG wire#powerrail
      "Control_05"(irTag := "Scaled_AI".GasAnalyzerCO, iiTag := "1DB_mirror_aiw".aiw_QT503b_CO, iouWarning := "Warning_DB".GasAnalyzerCO, iouAlarm := "Alarm_DB".GasAnalyzerCO, owCode => "1DB_AICode".GasAnalyzerCO, oxFault => "1DB_AICode".xF_QT503b_CO)
   END_RUNG
   // the same network as SCL:
   "Control_05"(irTag := "Scaled_AI".GasAnalyzerCO,   // "1FB_Control"
                iiTag := "1DB_mirror_aiw".aiw_QT503b_CO,
                iouWarning := "Warning_DB".GasAnalyzerCO,
                iouAlarm := "Alarm_DB".GasAnalyzerCO,
                owCode => "1DB_AICode".GasAnalyzerCO,
                oxFault => "1DB_AICode".xF_QT503b_CO);
END_REGION

REGION Network 6: Концентрация SO2 QT503b_SO2
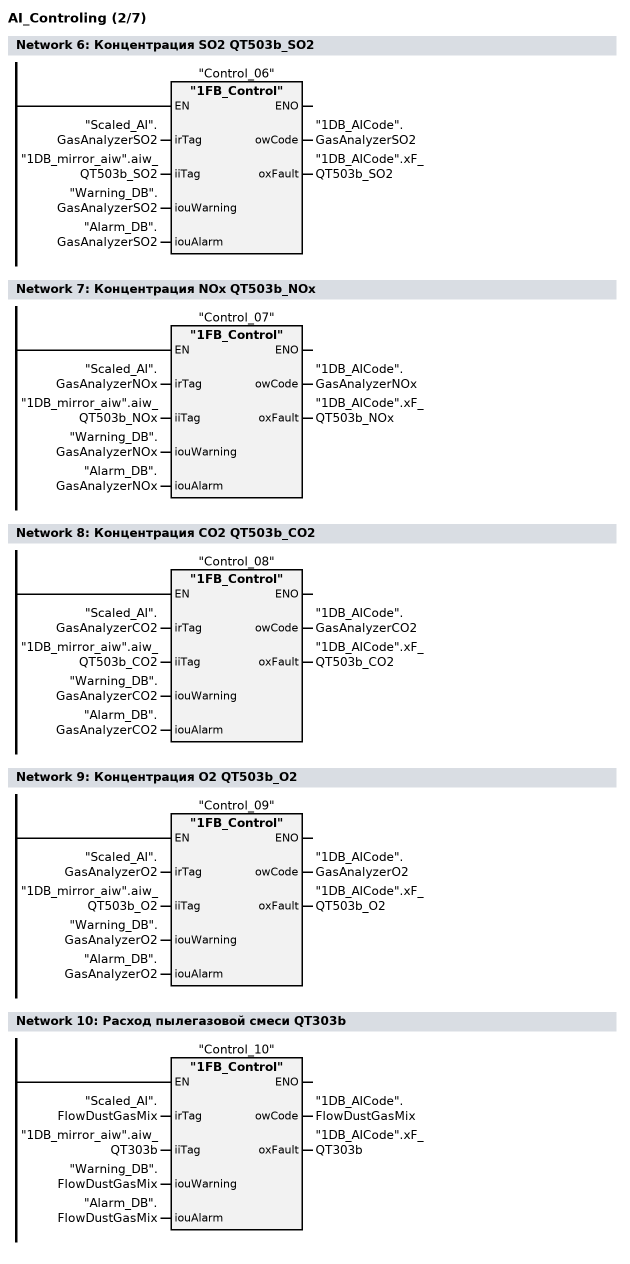
   RUNG wire#powerrail
      "Control_06"(irTag := "Scaled_AI".GasAnalyzerSO2, iiTag := "1DB_mirror_aiw".aiw_QT503b_SO2, iouWarning := "Warning_DB".GasAnalyzerSO2, iouAlarm := "Alarm_DB".GasAnalyzerSO2, owCode => "1DB_AICode".GasAnalyzerSO2, oxFault => "1DB_AICode".xF_QT503b_SO2)
   END_RUNG
   // the same network as SCL:
   "Control_06"(irTag := "Scaled_AI".GasAnalyzerSO2,   // "1FB_Control"
                iiTag := "1DB_mirror_aiw".aiw_QT503b_SO2,
                iouWarning := "Warning_DB".GasAnalyzerSO2,
                iouAlarm := "Alarm_DB".GasAnalyzerSO2,
                owCode => "1DB_AICode".GasAnalyzerSO2,
                oxFault => "1DB_AICode".xF_QT503b_SO2);
END_REGION

REGION Network 7: Концентрация NOx QT503b_NOx
   RUNG wire#powerrail
      "Control_07"(irTag := "Scaled_AI".GasAnalyzerNOx, iiTag := "1DB_mirror_aiw".aiw_QT503b_NOx, iouWarning := "Warning_DB".GasAnalyzerNOx, iouAlarm := "Alarm_DB".GasAnalyzerNOx, owCode => "1DB_AICode".GasAnalyzerNOx, oxFault => "1DB_AICode".xF_QT503b_NOx)
   END_RUNG
   // the same network as SCL:
   "Control_07"(irTag := "Scaled_AI".GasAnalyzerNOx,   // "1FB_Control"
                iiTag := "1DB_mirror_aiw".aiw_QT503b_NOx,
                iouWarning := "Warning_DB".GasAnalyzerNOx,
                iouAlarm := "Alarm_DB".GasAnalyzerNOx,
                owCode => "1DB_AICode".GasAnalyzerNOx,
                oxFault => "1DB_AICode".xF_QT503b_NOx);
END_REGION

REGION Network 8: Концентрация CO2 QT503b_CO2
   RUNG wire#powerrail
      "Control_08"(irTag := "Scaled_AI".GasAnalyzerCO2, iiTag := "1DB_mirror_aiw".aiw_QT503b_CO2, iouWarning := "Warning_DB".GasAnalyzerCO2, iouAlarm := "Alarm_DB".GasAnalyzerCO2, owCode => "1DB_AICode".GasAnalyzerCO2, oxFault => "1DB_AICode".xF_QT503b_CO2)
   END_RUNG
   // the same network as SCL:
   "Control_08"(irTag := "Scaled_AI".GasAnalyzerCO2,   // "1FB_Control"
                iiTag := "1DB_mirror_aiw".aiw_QT503b_CO2,
                iouWarning := "Warning_DB".GasAnalyzerCO2,
                iouAlarm := "Alarm_DB".GasAnalyzerCO2,
                owCode => "1DB_AICode".GasAnalyzerCO2,
                oxFault => "1DB_AICode".xF_QT503b_CO2);
END_REGION

REGION Network 9: Концентрация O2 QT503b_O2
   RUNG wire#powerrail
      "Control_09"(irTag := "Scaled_AI".GasAnalyzerO2, iiTag := "1DB_mirror_aiw".aiw_QT503b_O2, iouWarning := "Warning_DB".GasAnalyzerO2, iouAlarm := "Alarm_DB".GasAnalyzerO2, owCode => "1DB_AICode".GasAnalyzerO2, oxFault => "1DB_AICode".xF_QT503b_O2)
   END_RUNG
   // the same network as SCL:
   "Control_09"(irTag := "Scaled_AI".GasAnalyzerO2,   // "1FB_Control"
                iiTag := "1DB_mirror_aiw".aiw_QT503b_O2,
                iouWarning := "Warning_DB".GasAnalyzerO2,
                iouAlarm := "Alarm_DB".GasAnalyzerO2,
                owCode => "1DB_AICode".GasAnalyzerO2,
                oxFault => "1DB_AICode".xF_QT503b_O2);
END_REGION

REGION Network 10: Расход пылегазовой смеси QT303b
   RUNG wire#powerrail
      "Control_10"(irTag := "Scaled_AI".FlowDustGasMix, iiTag := "1DB_mirror_aiw".aiw_QT303b, iouWarning := "Warning_DB".FlowDustGasMix, iouAlarm := "Alarm_DB".FlowDustGasMix, owCode => "1DB_AICode".FlowDustGasMix, oxFault => "1DB_AICode".xF_QT303b)
   END_RUNG
   // the same network as SCL:
   "Control_10"(irTag := "Scaled_AI".FlowDustGasMix,   // "1FB_Control"
                iiTag := "1DB_mirror_aiw".aiw_QT303b,
                iouWarning := "Warning_DB".FlowDustGasMix,
                iouAlarm := "Alarm_DB".FlowDustGasMix,
                owCode => "1DB_AICode".FlowDustGasMix,
                oxFault => "1DB_AICode".xF_QT303b);
END_REGION

REGION Network 11: Концентрация пыли QT403b
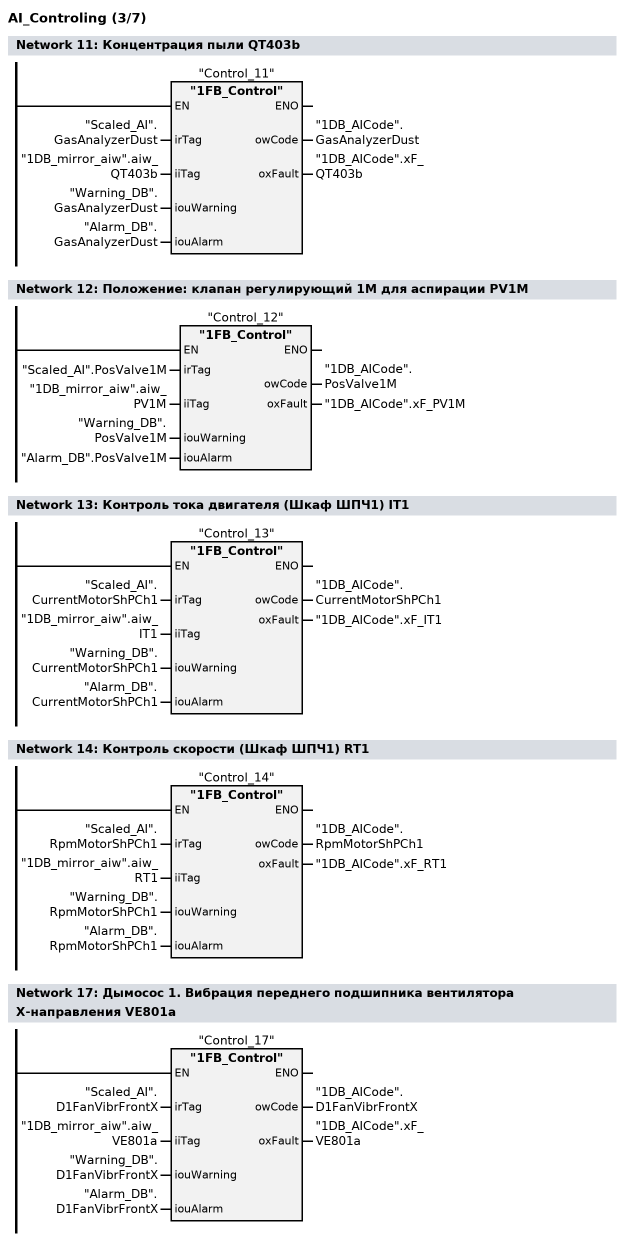
   RUNG wire#powerrail
      "Control_11"(irTag := "Scaled_AI".GasAnalyzerDust, iiTag := "1DB_mirror_aiw".aiw_QT403b, iouWarning := "Warning_DB".GasAnalyzerDust, iouAlarm := "Alarm_DB".GasAnalyzerDust, owCode => "1DB_AICode".GasAnalyzerDust, oxFault => "1DB_AICode".xF_QT403b)
   END_RUNG
   // the same network as SCL:
   "Control_11"(irTag := "Scaled_AI".GasAnalyzerDust,   // "1FB_Control"
                iiTag := "1DB_mirror_aiw".aiw_QT403b,
                iouWarning := "Warning_DB".GasAnalyzerDust,
                iouAlarm := "Alarm_DB".GasAnalyzerDust,
                owCode => "1DB_AICode".GasAnalyzerDust,
                oxFault => "1DB_AICode".xF_QT403b);
END_REGION

REGION Network 12: Положение: клапан регулирующий 1M для аспирации PV1M
   RUNG wire#powerrail
      "Control_12"(irTag := "Scaled_AI".PosValve1M, iiTag := "1DB_mirror_aiw".aiw_PV1M, iouWarning := "Warning_DB".PosValve1M, iouAlarm := "Alarm_DB".PosValve1M, owCode => "1DB_AICode".PosValve1M, oxFault => "1DB_AICode".xF_PV1M)
   END_RUNG
   // the same network as SCL:
   "Control_12"(irTag := "Scaled_AI".PosValve1M,   // "1FB_Control"
                iiTag := "1DB_mirror_aiw".aiw_PV1M,
                iouWarning := "Warning_DB".PosValve1M,
                iouAlarm := "Alarm_DB".PosValve1M,
                owCode => "1DB_AICode".PosValve1M,
                oxFault => "1DB_AICode".xF_PV1M);
END_REGION

REGION Network 13: Контроль тока двигателя (Шкаф ШПЧ1) IT1
   RUNG wire#powerrail
      "Control_13"(irTag := "Scaled_AI".CurrentMotorShPCh1, iiTag := "1DB_mirror_aiw".aiw_IT1, iouWarning := "Warning_DB".CurrentMotorShPCh1, iouAlarm := "Alarm_DB".CurrentMotorShPCh1, owCode => "1DB_AICode".CurrentMotorShPCh1, oxFault => "1DB_AICode".xF_IT1)
   END_RUNG
   // the same network as SCL:
   "Control_13"(irTag := "Scaled_AI".CurrentMotorShPCh1,   // "1FB_Control"
                iiTag := "1DB_mirror_aiw".aiw_IT1,
                iouWarning := "Warning_DB".CurrentMotorShPCh1,
                iouAlarm := "Alarm_DB".CurrentMotorShPCh1,
                owCode => "1DB_AICode".CurrentMotorShPCh1,
                oxFault => "1DB_AICode".xF_IT1);
END_REGION

REGION Network 14: Контроль скорости (Шкаф ШПЧ1) RT1
   RUNG wire#powerrail
      "Control_14"(irTag := "Scaled_AI".RpmMotorShPCh1, iiTag := "1DB_mirror_aiw".aiw_RT1, iouWarning := "Warning_DB".RpmMotorShPCh1, iouAlarm := "Alarm_DB".RpmMotorShPCh1, owCode => "1DB_AICode".RpmMotorShPCh1, oxFault => "1DB_AICode".xF_RT1)
   END_RUNG
   // the same network as SCL:
   "Control_14"(irTag := "Scaled_AI".RpmMotorShPCh1,   // "1FB_Control"
                iiTag := "1DB_mirror_aiw".aiw_RT1,
                iouWarning := "Warning_DB".RpmMotorShPCh1,
                iouAlarm := "Alarm_DB".RpmMotorShPCh1,
                owCode => "1DB_AICode".RpmMotorShPCh1,
                oxFault => "1DB_AICode".xF_RT1);
END_REGION

REGION Network 15: 2 резервных места
END_REGION

REGION Network 16: 2 резервных места
END_REGION

REGION Network 17: Дымосос 1. Вибрация переднего подшипника вентилятора X-направления VE801a
   RUNG wire#powerrail
      "Control_17"(irTag := "Scaled_AI".D1FanVibrFrontX, iiTag := "1DB_mirror_aiw".aiw_VE801a, iouWarning := "Warning_DB".D1FanVibrFrontX, iouAlarm := "Alarm_DB".D1FanVibrFrontX, owCode => "1DB_AICode".D1FanVibrFrontX, oxFault => "1DB_AICode".xF_VE801a)
   END_RUNG
   // the same network as SCL:
   "Control_17"(irTag := "Scaled_AI".D1FanVibrFrontX,   // "1FB_Control"
                iiTag := "1DB_mirror_aiw".aiw_VE801a,
                iouWarning := "Warning_DB".D1FanVibrFrontX,
                iouAlarm := "Alarm_DB".D1FanVibrFrontX,
                owCode => "1DB_AICode".D1FanVibrFrontX,
                oxFault => "1DB_AICode".xF_VE801a);
END_REGION

REGION Network 18: Дымосос 1. Вибрация переднего подшипника вентилятора Y-направления VE802a
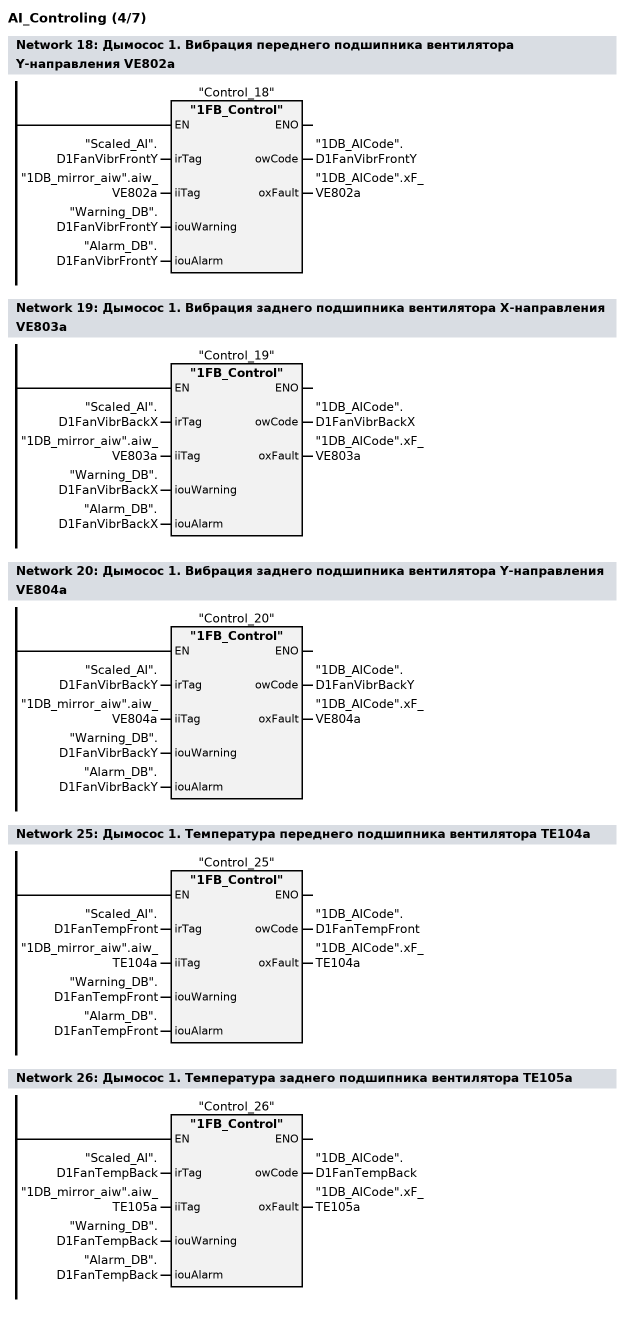
   RUNG wire#powerrail
      "Control_18"(irTag := "Scaled_AI".D1FanVibrFrontY, iiTag := "1DB_mirror_aiw".aiw_VE802a, iouWarning := "Warning_DB".D1FanVibrFrontY, iouAlarm := "Alarm_DB".D1FanVibrFrontY, owCode => "1DB_AICode".D1FanVibrFrontY, oxFault => "1DB_AICode".xF_VE802a)
   END_RUNG
   // the same network as SCL:
   "Control_18"(irTag := "Scaled_AI".D1FanVibrFrontY,   // "1FB_Control"
                iiTag := "1DB_mirror_aiw".aiw_VE802a,
                iouWarning := "Warning_DB".D1FanVibrFrontY,
                iouAlarm := "Alarm_DB".D1FanVibrFrontY,
                owCode => "1DB_AICode".D1FanVibrFrontY,
                oxFault => "1DB_AICode".xF_VE802a);
END_REGION

REGION Network 19: Дымосос 1. Вибрация заднего подшипника вентилятора X-направления VE803a
   RUNG wire#powerrail
      "Control_19"(irTag := "Scaled_AI".D1FanVibrBackX, iiTag := "1DB_mirror_aiw".aiw_VE803a, iouWarning := "Warning_DB".D1FanVibrBackX, iouAlarm := "Alarm_DB".D1FanVibrBackX, owCode => "1DB_AICode".D1FanVibrBackX, oxFault => "1DB_AICode".xF_VE803a)
   END_RUNG
   // the same network as SCL:
   "Control_19"(irTag := "Scaled_AI".D1FanVibrBackX,   // "1FB_Control"
                iiTag := "1DB_mirror_aiw".aiw_VE803a,
                iouWarning := "Warning_DB".D1FanVibrBackX,
                iouAlarm := "Alarm_DB".D1FanVibrBackX,
                owCode => "1DB_AICode".D1FanVibrBackX,
                oxFault => "1DB_AICode".xF_VE803a);
END_REGION

REGION Network 20: Дымосос 1. Вибрация заднего подшипника вентилятора Y-направления VE804a
   RUNG wire#powerrail
      "Control_20"(irTag := "Scaled_AI".D1FanVibrBackY, iiTag := "1DB_mirror_aiw".aiw_VE804a, iouWarning := "Warning_DB".D1FanVibrBackY, iouAlarm := "Alarm_DB".D1FanVibrBackY, owCode => "1DB_AICode".D1FanVibrBackY, oxFault => "1DB_AICode".xF_VE804a)
   END_RUNG
   // the same network as SCL:
   "Control_20"(irTag := "Scaled_AI".D1FanVibrBackY,   // "1FB_Control"
                iiTag := "1DB_mirror_aiw".aiw_VE804a,
                iouWarning := "Warning_DB".D1FanVibrBackY,
                iouAlarm := "Alarm_DB".D1FanVibrBackY,
                owCode => "1DB_AICode".D1FanVibrBackY,
                oxFault => "1DB_AICode".xF_VE804a);
END_REGION

REGION Network 21: 4 резервных места
END_REGION

REGION Network 22: 4 резервных места
END_REGION

REGION Network 23: 4 резервных места
END_REGION

REGION Network 24: 4 резервных места
END_REGION

REGION Network 25: Дымосос 1. Температура переднего подшипника вентилятора TE104a
   RUNG wire#powerrail
      "Control_25"(irTag := "Scaled_AI".D1FanTempFront, iiTag := "1DB_mirror_aiw".aiw_TE104a, iouWarning := "Warning_DB".D1FanTempFront, iouAlarm := "Alarm_DB".D1FanTempFront, owCode => "1DB_AICode".D1FanTempFront, oxFault => "1DB_AICode".xF_TE104a)
   END_RUNG
   // the same network as SCL:
   "Control_25"(irTag := "Scaled_AI".D1FanTempFront,   // "1FB_Control"
                iiTag := "1DB_mirror_aiw".aiw_TE104a,
                iouWarning := "Warning_DB".D1FanTempFront,
                iouAlarm := "Alarm_DB".D1FanTempFront,
                owCode => "1DB_AICode".D1FanTempFront,
                oxFault => "1DB_AICode".xF_TE104a);
END_REGION

REGION Network 26: Дымосос 1. Температура заднего подшипника вентилятора TE105a
   RUNG wire#powerrail
      "Control_26"(irTag := "Scaled_AI".D1FanTempBack, iiTag := "1DB_mirror_aiw".aiw_TE105a, iouWarning := "Warning_DB".D1FanTempBack, iouAlarm := "Alarm_DB".D1FanTempBack, owCode => "1DB_AICode".D1FanTempBack, oxFault => "1DB_AICode".xF_TE105a)
   END_RUNG
   // the same network as SCL:
   "Control_26"(irTag := "Scaled_AI".D1FanTempBack,   // "1FB_Control"
                iiTag := "1DB_mirror_aiw".aiw_TE105a,
                iouWarning := "Warning_DB".D1FanTempBack,
                iouAlarm := "Alarm_DB".D1FanTempBack,
                owCode => "1DB_AICode".D1FanTempBack,
                oxFault => "1DB_AICode".xF_TE105a);
END_REGION

REGION Network 27: Электродвигатель дымососа 1. Температура переднего подшипника TE106a
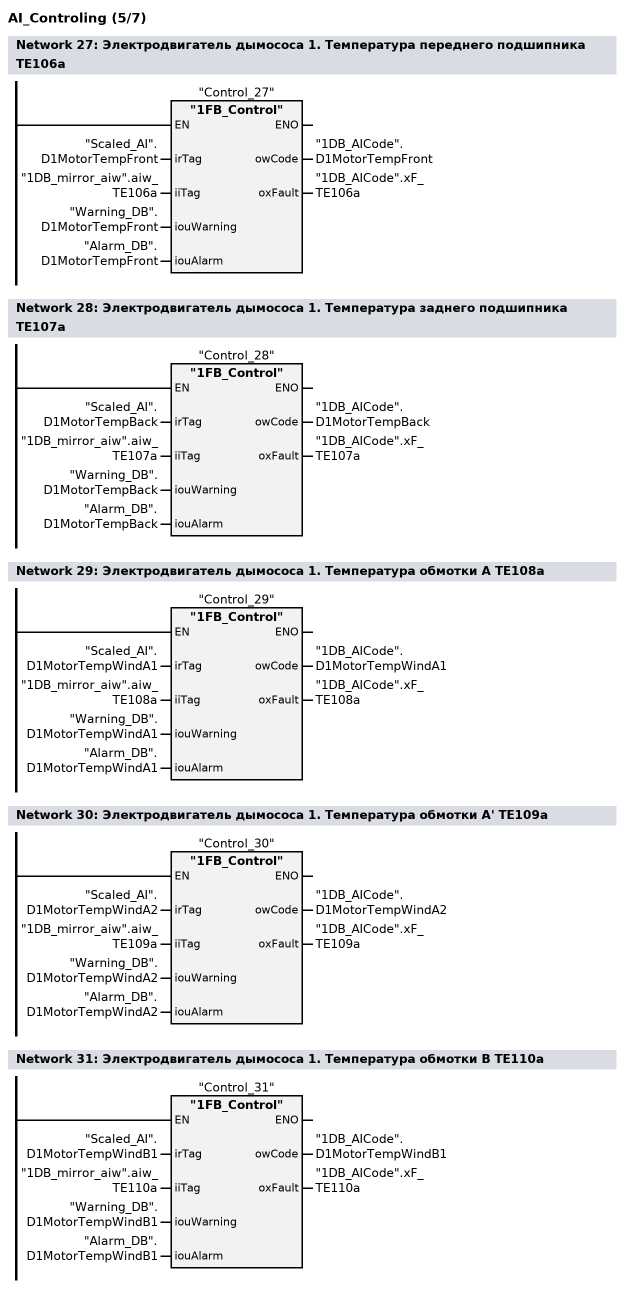
   RUNG wire#powerrail
      "Control_27"(irTag := "Scaled_AI".D1MotorTempFront, iiTag := "1DB_mirror_aiw".aiw_TE106a, iouWarning := "Warning_DB".D1MotorTempFront, iouAlarm := "Alarm_DB".D1MotorTempFront, owCode => "1DB_AICode".D1MotorTempFront, oxFault => "1DB_AICode".xF_TE106a)
   END_RUNG
   // the same network as SCL:
   "Control_27"(irTag := "Scaled_AI".D1MotorTempFront,   // "1FB_Control"
                iiTag := "1DB_mirror_aiw".aiw_TE106a,
                iouWarning := "Warning_DB".D1MotorTempFront,
                iouAlarm := "Alarm_DB".D1MotorTempFront,
                owCode => "1DB_AICode".D1MotorTempFront,
                oxFault => "1DB_AICode".xF_TE106a);
END_REGION

REGION Network 28: Электродвигатель дымососа 1. Температура заднего подшипника TE107a
   RUNG wire#powerrail
      "Control_28"(irTag := "Scaled_AI".D1MotorTempBack, iiTag := "1DB_mirror_aiw".aiw_TE107a, iouWarning := "Warning_DB".D1MotorTempBack, iouAlarm := "Alarm_DB".D1MotorTempBack, owCode => "1DB_AICode".D1MotorTempBack, oxFault => "1DB_AICode".xF_TE107a)
   END_RUNG
   // the same network as SCL:
   "Control_28"(irTag := "Scaled_AI".D1MotorTempBack,   // "1FB_Control"
                iiTag := "1DB_mirror_aiw".aiw_TE107a,
                iouWarning := "Warning_DB".D1MotorTempBack,
                iouAlarm := "Alarm_DB".D1MotorTempBack,
                owCode => "1DB_AICode".D1MotorTempBack,
                oxFault => "1DB_AICode".xF_TE107a);
END_REGION

REGION Network 29: Электродвигатель дымососа 1. Температура обмотки А TE108a
   RUNG wire#powerrail
      "Control_29"(irTag := "Scaled_AI".D1MotorTempWindA1, iiTag := "1DB_mirror_aiw".aiw_TE108a, iouWarning := "Warning_DB".D1MotorTempWindA1, iouAlarm := "Alarm_DB".D1MotorTempWindA1, owCode => "1DB_AICode".D1MotorTempWindA1, oxFault => "1DB_AICode".xF_TE108a)
   END_RUNG
   // the same network as SCL:
   "Control_29"(irTag := "Scaled_AI".D1MotorTempWindA1,   // "1FB_Control"
                iiTag := "1DB_mirror_aiw".aiw_TE108a,
                iouWarning := "Warning_DB".D1MotorTempWindA1,
                iouAlarm := "Alarm_DB".D1MotorTempWindA1,
                owCode => "1DB_AICode".D1MotorTempWindA1,
                oxFault => "1DB_AICode".xF_TE108a);
END_REGION

REGION Network 30: Электродвигатель дымососа 1. Температура обмотки А' TE109a
   RUNG wire#powerrail
      "Control_30"(irTag := "Scaled_AI".D1MotorTempWindA2, iiTag := "1DB_mirror_aiw".aiw_TE109a, iouWarning := "Warning_DB".D1MotorTempWindA2, iouAlarm := "Alarm_DB".D1MotorTempWindA2, owCode => "1DB_AICode".D1MotorTempWindA2, oxFault => "1DB_AICode".xF_TE109a)
   END_RUNG
   // the same network as SCL:
   "Control_30"(irTag := "Scaled_AI".D1MotorTempWindA2,   // "1FB_Control"
                iiTag := "1DB_mirror_aiw".aiw_TE109a,
                iouWarning := "Warning_DB".D1MotorTempWindA2,
                iouAlarm := "Alarm_DB".D1MotorTempWindA2,
                owCode => "1DB_AICode".D1MotorTempWindA2,
                oxFault => "1DB_AICode".xF_TE109a);
END_REGION

REGION Network 31: Электродвигатель дымососа 1. Температура обмотки B TE110a
   RUNG wire#powerrail
      "Control_31"(irTag := "Scaled_AI".D1MotorTempWindB1, iiTag := "1DB_mirror_aiw".aiw_TE110a, iouWarning := "Warning_DB".D1MotorTempWindB1, iouAlarm := "Alarm_DB".D1MotorTempWindB1, owCode => "1DB_AICode".D1MotorTempWindB1, oxFault => "1DB_AICode".xF_TE110a)
   END_RUNG
   // the same network as SCL:
   "Control_31"(irTag := "Scaled_AI".D1MotorTempWindB1,   // "1FB_Control"
                iiTag := "1DB_mirror_aiw".aiw_TE110a,
                iouWarning := "Warning_DB".D1MotorTempWindB1,
                iouAlarm := "Alarm_DB".D1MotorTempWindB1,
                owCode => "1DB_AICode".D1MotorTempWindB1,
                oxFault => "1DB_AICode".xF_TE110a);
END_REGION

REGION Network 32: Электродвигатель дымососа 1. Температура обмотки B' TE111a
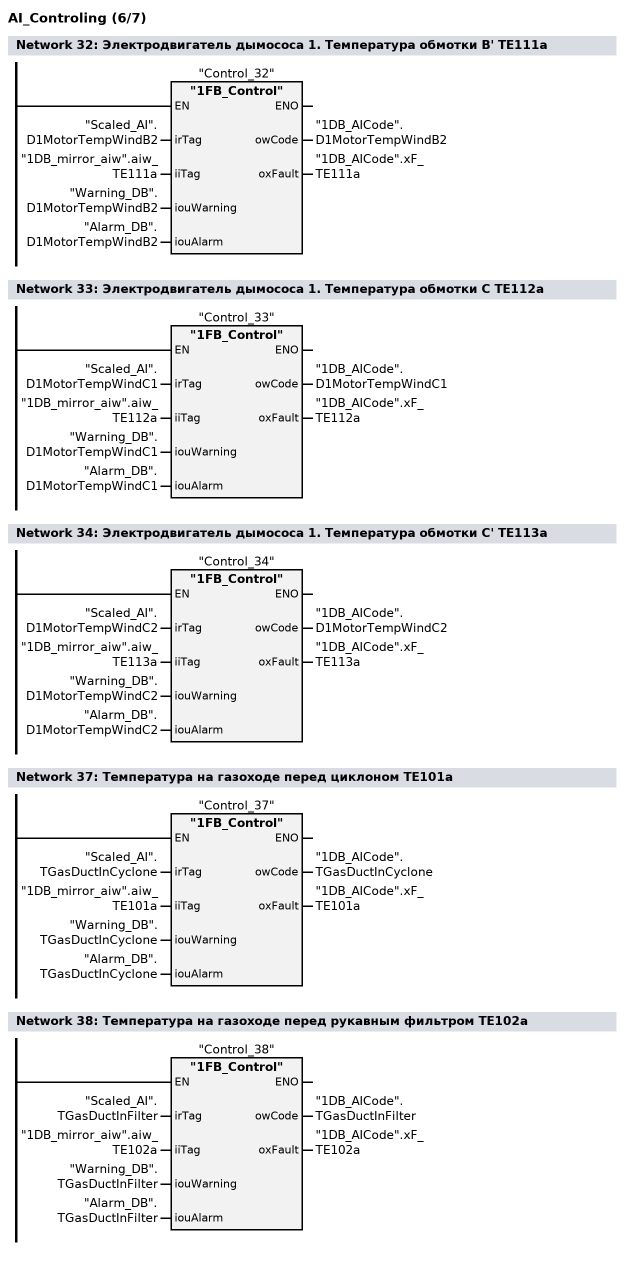
   RUNG wire#powerrail
      "Control_32"(irTag := "Scaled_AI".D1MotorTempWindB2, iiTag := "1DB_mirror_aiw".aiw_TE111a, iouWarning := "Warning_DB".D1MotorTempWindB2, iouAlarm := "Alarm_DB".D1MotorTempWindB2, owCode => "1DB_AICode".D1MotorTempWindB2, oxFault => "1DB_AICode".xF_TE111a)
   END_RUNG
   // the same network as SCL:
   "Control_32"(irTag := "Scaled_AI".D1MotorTempWindB2,   // "1FB_Control"
                iiTag := "1DB_mirror_aiw".aiw_TE111a,
                iouWarning := "Warning_DB".D1MotorTempWindB2,
                iouAlarm := "Alarm_DB".D1MotorTempWindB2,
                owCode => "1DB_AICode".D1MotorTempWindB2,
                oxFault => "1DB_AICode".xF_TE111a);
END_REGION

REGION Network 33: Электродвигатель дымососа 1. Температура обмотки C TE112a
   RUNG wire#powerrail
      "Control_33"(irTag := "Scaled_AI".D1MotorTempWindC1, iiTag := "1DB_mirror_aiw".aiw_TE112a, iouWarning := "Warning_DB".D1MotorTempWindC1, iouAlarm := "Alarm_DB".D1MotorTempWindC1, owCode => "1DB_AICode".D1MotorTempWindC1, oxFault => "1DB_AICode".xF_TE112a)
   END_RUNG
   // the same network as SCL:
   "Control_33"(irTag := "Scaled_AI".D1MotorTempWindC1,   // "1FB_Control"
                iiTag := "1DB_mirror_aiw".aiw_TE112a,
                iouWarning := "Warning_DB".D1MotorTempWindC1,
                iouAlarm := "Alarm_DB".D1MotorTempWindC1,
                owCode => "1DB_AICode".D1MotorTempWindC1,
                oxFault => "1DB_AICode".xF_TE112a);
END_REGION

REGION Network 34: Электродвигатель дымососа 1. Температура обмотки C' TE113a
   RUNG wire#powerrail
      "Control_34"(irTag := "Scaled_AI".D1MotorTempWindC2, iiTag := "1DB_mirror_aiw".aiw_TE113a, iouWarning := "Warning_DB".D1MotorTempWindC2, iouAlarm := "Alarm_DB".D1MotorTempWindC2, owCode => "1DB_AICode".D1MotorTempWindC2, oxFault => "1DB_AICode".xF_TE113a)
   END_RUNG
   // the same network as SCL:
   "Control_34"(irTag := "Scaled_AI".D1MotorTempWindC2,   // "1FB_Control"
                iiTag := "1DB_mirror_aiw".aiw_TE113a,
                iouWarning := "Warning_DB".D1MotorTempWindC2,
                iouAlarm := "Alarm_DB".D1MotorTempWindC2,
                owCode => "1DB_AICode".D1MotorTempWindC2,
                oxFault => "1DB_AICode".xF_TE113a);
END_REGION

REGION Network 35: 2 резервных места
END_REGION

REGION Network 36: 2 резервных места
END_REGION

REGION Network 37: Температура на газоходе перед циклоном TE101a
   RUNG wire#powerrail
      "Control_37"(irTag := "Scaled_AI".TGasDuctInCyclone, iiTag := "1DB_mirror_aiw".aiw_TE101a, iouWarning := "Warning_DB".TGasDuctInCyclone, iouAlarm := "Alarm_DB".TGasDuctInCyclone, owCode => "1DB_AICode".TGasDuctInCyclone, oxFault => "1DB_AICode".xF_TE101a)
   END_RUNG
   // the same network as SCL:
   "Control_37"(irTag := "Scaled_AI".TGasDuctInCyclone,   // "1FB_Control"
                iiTag := "1DB_mirror_aiw".aiw_TE101a,
                iouWarning := "Warning_DB".TGasDuctInCyclone,
                iouAlarm := "Alarm_DB".TGasDuctInCyclone,
                owCode => "1DB_AICode".TGasDuctInCyclone,
                oxFault => "1DB_AICode".xF_TE101a);
END_REGION

REGION Network 38: Температура на газоходе перед рукавным фильтром TE102a
   RUNG wire#powerrail
      "Control_38"(irTag := "Scaled_AI".TGasDuctInFilter, iiTag := "1DB_mirror_aiw".aiw_TE102a, iouWarning := "Warning_DB".TGasDuctInFilter, iouAlarm := "Alarm_DB".TGasDuctInFilter, owCode => "1DB_AICode".TGasDuctInFilter, oxFault => "1DB_AICode".xF_TE102a)
   END_RUNG
   // the same network as SCL:
   "Control_38"(irTag := "Scaled_AI".TGasDuctInFilter,   // "1FB_Control"
                iiTag := "1DB_mirror_aiw".aiw_TE102a,
                iouWarning := "Warning_DB".TGasDuctInFilter,
                iouAlarm := "Alarm_DB".TGasDuctInFilter,
                owCode => "1DB_AICode".TGasDuctInFilter,
                oxFault => "1DB_AICode".xF_TE102a);
END_REGION

REGION Network 39: Температура газа на выходе из трубы TE103a
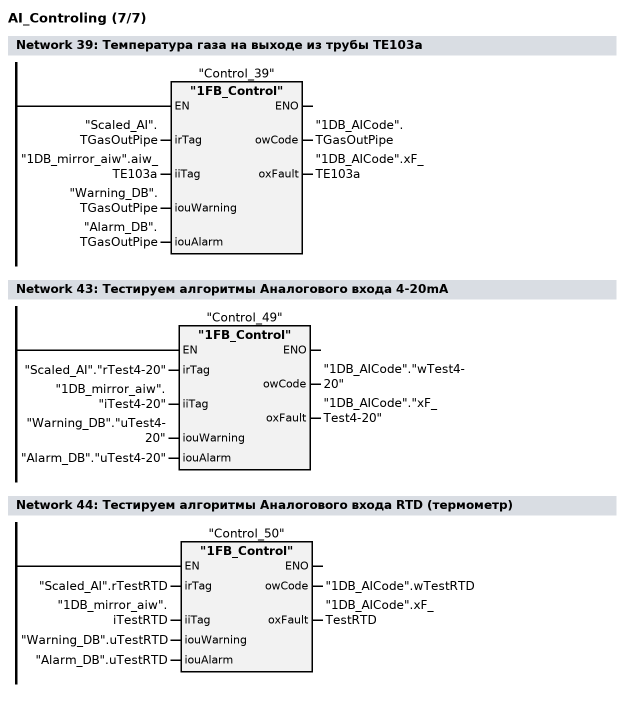
   RUNG wire#powerrail
      "Control_39"(irTag := "Scaled_AI".TGasOutPipe, iiTag := "1DB_mirror_aiw".aiw_TE103a, iouWarning := "Warning_DB".TGasOutPipe, iouAlarm := "Alarm_DB".TGasOutPipe, owCode => "1DB_AICode".TGasOutPipe, oxFault => "1DB_AICode".xF_TE103a)
   END_RUNG
   // the same network as SCL:
   "Control_39"(irTag := "Scaled_AI".TGasOutPipe,   // "1FB_Control"
                iiTag := "1DB_mirror_aiw".aiw_TE103a,
                iouWarning := "Warning_DB".TGasOutPipe,
                iouAlarm := "Alarm_DB".TGasOutPipe,
                owCode => "1DB_AICode".TGasOutPipe,
                oxFault => "1DB_AICode".xF_TE103a);
END_REGION

REGION Network 43: Тестируем алгоритмы Аналогового входа 4-20mA
   RUNG wire#powerrail
      "Control_49"(irTag := "Scaled_AI"."rTest4-20", iiTag := "1DB_mirror_aiw"."iTest4-20", iouWarning := "Warning_DB"."uTest4-20", iouAlarm := "Alarm_DB"."uTest4-20", owCode => "1DB_AICode"."wTest4-20", oxFault => "1DB_AICode"."xF_Test4-20")
   END_RUNG
   // the same network as SCL:
   "Control_49"(irTag := "Scaled_AI"."rTest4-20",   // "1FB_Control"
                iiTag := "1DB_mirror_aiw"."iTest4-20",
                iouWarning := "Warning_DB"."uTest4-20",
                iouAlarm := "Alarm_DB"."uTest4-20",
                owCode => "1DB_AICode"."wTest4-20",
                oxFault => "1DB_AICode"."xF_Test4-20");
END_REGION

REGION Network 44: Тестируем алгоритмы Аналогового входа RTD (термометр)
   RUNG wire#powerrail
      "Control_50"(irTag := "Scaled_AI".rTestRTD, iiTag := "1DB_mirror_aiw".iTestRTD, iouWarning := "Warning_DB".uTestRTD, iouAlarm := "Alarm_DB".uTestRTD, owCode => "1DB_AICode".wTestRTD, oxFault => "1DB_AICode".xF_TestRTD)
   END_RUNG
   // the same network as SCL:
   "Control_50"(irTag := "Scaled_AI".rTestRTD,   // "1FB_Control"
                iiTag := "1DB_mirror_aiw".iTestRTD,
                iouWarning := "Warning_DB".uTestRTD,
                iouAlarm := "Alarm_DB".uTestRTD,
                owCode => "1DB_AICode".wTestRTD,
                oxFault => "1DB_AICode".xF_TestRTD);
END_REGION
END_FUNCTION

// folder: Shadow

FUNCTION "1FC_CONFIGs" : Void   // FC500, LAD
{ S7_Optimized_Access := 'TRUE' }
VERSION : 0.1
   VAR_TEMP
      txSave : Bool;   // Сохранить
      txRestore : Bool;   // Возобновить
      wRet_Val_Save : Word;   // Код ошибки
      wRet_Val_Restore : Word;   // Код ошибки
   END_VAR
   VAR_TEMP   // added for the SCL form of the ladder/FBD networks
      _w1 : Bool;
   END_VAR
BEGIN

REGION Network 2: Сохранить
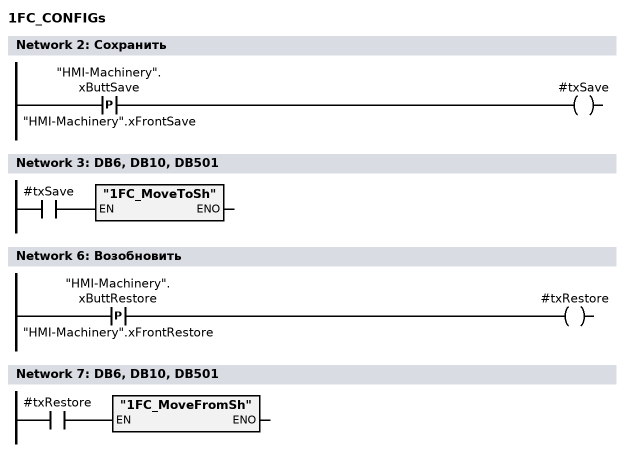
   RUNG wire#powerrail
      P_Contact(operand := "HMI-Machinery".xButtSave, bit := "HMI-Machinery".xFrontSave)
      Coil( #txSave )
   END_RUNG
   // the same network as SCL:
   #_w1 := "HMI-Machinery".xButtSave AND NOT "HMI-Machinery".xFrontSave;   // rising edge of "HMI-Machinery".xButtSave
   "HMI-Machinery".xFrontSave := "HMI-Machinery".xButtSave;
   #txSave := #_w1;
END_REGION

REGION Network 3: DB6, DB10, DB501
   RUNG wire#powerrail
      Contact( #txSave )
      "1FC_MoveToSh"()
   END_RUNG
   // the same network as SCL:
   IF #txSave THEN "1FC_MoveToSh"(); END_IF;
END_REGION

REGION Network 6: Возобновить
   RUNG wire#powerrail
      P_Contact(operand := "HMI-Machinery".xButtRestore, bit := "HMI-Machinery".xFrontRestore)
      Coil( #txRestore )
   END_RUNG
   // the same network as SCL:
   #_w1 := "HMI-Machinery".xButtRestore AND NOT "HMI-Machinery".xFrontRestore;   // rising edge of "HMI-Machinery".xButtRestore
   "HMI-Machinery".xFrontRestore := "HMI-Machinery".xButtRestore;
   #txRestore := #_w1;
END_REGION

REGION Network 7: DB6, DB10, DB501
   RUNG wire#powerrail
      Contact( #txRestore )
      "1FC_MoveFromSh"()
   END_RUNG
   // the same network as SCL:
   IF #txRestore THEN "1FC_MoveFromSh"(); END_IF;
END_REGION
END_FUNCTION

FUNCTION "1FC_MoveToSh" : Void   // FC501, SCL
{ S7_Optimized_Access := 'TRUE' }
VERSION : 0.1
BEGIN

   "1DB_AIConfig_Sh".RarefactFlueInCyclone := "1DB_AIConfig".RarefactFlueInCyclone;    "Alarm_DB_Sh".RarefactFlueInCyclone := "Alarm_DB".RarefactFlueInCyclone;
   "1DB_AIConfig_Sh".RarefactFlueInFilter :=  "1DB_AIConfig".RarefactFlueInFilter;     "Alarm_DB_Sh".RarefactFlueInFilter :=  "Alarm_DB".RarefactFlueInFilter;
   "1DB_AIConfig_Sh".RarefactFlueOutFilter := "1DB_AIConfig".RarefactFlueOutFilter;    "Alarm_DB_Sh".RarefactFlueOutFilter := "Alarm_DB".RarefactFlueOutFilter;
   "1DB_AIConfig_Sh".PressureComprAir := "1DB_AIConfig".PressureComprAir;  "Alarm_DB_Sh".PressureComprAir := "Alarm_DB".PressureComprAir;
   "1DB_AIConfig_Sh".GasAnalyzerCO :=    "1DB_AIConfig".GasAnalyzerCO;     "Alarm_DB_Sh".GasAnalyzerCO :=    "Alarm_DB".GasAnalyzerCO;
   "1DB_AIConfig_Sh".GasAnalyzerSO2 :=   "1DB_AIConfig".GasAnalyzerSO2;    "Alarm_DB_Sh".GasAnalyzerSO2 :=   "Alarm_DB".GasAnalyzerSO2;
   "1DB_AIConfig_Sh".GasAnalyzerNOx :=   "1DB_AIConfig".GasAnalyzerNOx;    "Alarm_DB_Sh".GasAnalyzerNOx :=   "Alarm_DB".GasAnalyzerNOx;
   "1DB_AIConfig_Sh".GasAnalyzerCO2 :=   "1DB_AIConfig".GasAnalyzerCO2;    "Alarm_DB_Sh".GasAnalyzerCO2 :=   "Alarm_DB".GasAnalyzerCO2;
   "1DB_AIConfig_Sh".GasAnalyzerO2 :=    "1DB_AIConfig".GasAnalyzerO2;     "Alarm_DB_Sh".GasAnalyzerO2 :=    "Alarm_DB".GasAnalyzerO2;
   "1DB_AIConfig_Sh".FlowDustGasMix :=   "1DB_AIConfig".FlowDustGasMix;    "Alarm_DB_Sh".FlowDustGasMix :=   "Alarm_DB".FlowDustGasMix;
   "1DB_AIConfig_Sh".GasAnalyzerDust :=  "1DB_AIConfig".GasAnalyzerDust;   "Alarm_DB_Sh".GasAnalyzerDust :=  "Alarm_DB".GasAnalyzerDust;
   "1DB_AIConfig_Sh".PosValve1M :=       "1DB_AIConfig".PosValve1M;        "Alarm_DB_Sh".PosValve1M :=       "Alarm_DB".PosValve1M;
   "1DB_AIConfig_Sh".CurrentMotorShPCh1 :=    "1DB_AIConfig".CurrentMotorShPCh1;       "Alarm_DB_Sh".CurrentMotorShPCh1 := "Alarm_DB".CurrentMotorShPCh1;
   "1DB_AIConfig_Sh".RpmMotorShPCh1 :=   "1DB_AIConfig".RpmMotorShPCh1;    "Alarm_DB_Sh".RpmMotorShPCh1 :=   "Alarm_DB".RpmMotorShPCh1;
   "1DB_AIConfig_Sh".D1FanVibrFrontX :=  "1DB_AIConfig".D1FanVibrFrontX;   "Alarm_DB_Sh".D1FanVibrFrontX :=  "Alarm_DB".D1FanVibrFrontX;
   "1DB_AIConfig_Sh".D1FanVibrFrontY :=  "1DB_AIConfig".D1FanVibrFrontY;   "Alarm_DB_Sh".D1FanVibrFrontY :=  "Alarm_DB".D1FanVibrFrontY;
   "1DB_AIConfig_Sh".D1FanVibrBackX :=   "1DB_AIConfig".D1FanVibrBackX;    "Alarm_DB_Sh".D1FanVibrBackX :=   "Alarm_DB".D1FanVibrBackX;
   "1DB_AIConfig_Sh".D1FanVibrBackY :=   "1DB_AIConfig".D1FanVibrBackY;    "Alarm_DB_Sh".D1FanVibrBackY :=   "Alarm_DB".D1FanVibrBackY;
   "1DB_AIConfig_Sh".D1FanTempFront :=   "1DB_AIConfig".D1FanTempFront;    "Alarm_DB_Sh".D1FanTempFront :=   "Alarm_DB".D1FanTempFront;
   "1DB_AIConfig_Sh".D1FanTempBack :=    "1DB_AIConfig".D1FanTempBack;     "Alarm_DB_Sh".D1FanTempBack :=    "Alarm_DB".D1FanTempBack;
   "1DB_AIConfig_Sh".D1MotorTempFront := "1DB_AIConfig".D1MotorTempFront;  "Alarm_DB_Sh".D1MotorTempFront := "Alarm_DB".D1MotorTempFront;
   "1DB_AIConfig_Sh".D1MotorTempBack :=  "1DB_AIConfig".D1MotorTempBack;   "Alarm_DB_Sh".D1MotorTempBack :=  "Alarm_DB".D1MotorTempBack;
   "1DB_AIConfig_Sh".D1MotorTempWindA1:= "1DB_AIConfig".D1MotorTempWindA1; "Alarm_DB_Sh".D1MotorTempWindA1:= "Alarm_DB".D1MotorTempWindA1;
   "1DB_AIConfig_Sh".D1MotorTempWindA2:= "1DB_AIConfig".D1MotorTempWindA2; "Alarm_DB_Sh".D1MotorTempWindA2:= "Alarm_DB".D1MotorTempWindA2;
   "1DB_AIConfig_Sh".D1MotorTempWindB1:= "1DB_AIConfig".D1MotorTempWindB1; "Alarm_DB_Sh".D1MotorTempWindB1:= "Alarm_DB".D1MotorTempWindB1;
   "1DB_AIConfig_Sh".D1MotorTempWindB2:= "1DB_AIConfig".D1MotorTempWindB2; "Alarm_DB_Sh".D1MotorTempWindB2:= "Alarm_DB".D1MotorTempWindB2;
   "1DB_AIConfig_Sh".D1MotorTempWindC1:= "1DB_AIConfig".D1MotorTempWindC1; "Alarm_DB_Sh".D1MotorTempWindC1:= "Alarm_DB".D1MotorTempWindC1;
   "1DB_AIConfig_Sh".D1MotorTempWindC2:= "1DB_AIConfig".D1MotorTempWindC2; "Alarm_DB_Sh".D1MotorTempWindC2:= "Alarm_DB".D1MotorTempWindC2;
   "1DB_AIConfig_Sh".TGasDuctInCyclone:= "1DB_AIConfig".TGasDuctInCyclone; "Alarm_DB_Sh".TGasDuctInCyclone:= "Alarm_DB".TGasDuctInCyclone;
   "1DB_AIConfig_Sh".TGasDuctInFilter := "1DB_AIConfig".TGasDuctInFilter;  "Alarm_DB_Sh".TGasDuctInFilter := "Alarm_DB".TGasDuctInFilter;
   "1DB_AIConfig_Sh".TGasOutPipe :=      "1DB_AIConfig".TGasOutPipe;       "Alarm_DB_Sh".TGasOutPipe :=      "Alarm_DB".TGasOutPipe;

   "HMI-Machinery_Sh"."1M_PID" := "HMI-Machinery"."1M_PID";
   "HMI-Machinery_Sh".Dym_PID :=  "HMI-Machinery".Dym_PID;
END_FUNCTION

FUNCTION "1FC_MoveFromSh" : Void   // FC502, SCL
{ S7_Optimized_Access := 'TRUE' }
VERSION : 0.1
BEGIN

   "1DB_AIConfig".RarefactFlueInCyclone := "1DB_AIConfig_Sh".RarefactFlueInCyclone;    "Alarm_DB".RarefactFlueInCyclone := "Alarm_DB_Sh".RarefactFlueInCyclone;
   "1DB_AIConfig".RarefactFlueInFilter :=  "1DB_AIConfig_Sh".RarefactFlueInFilter;     "Alarm_DB".RarefactFlueInFilter :=  "Alarm_DB_Sh".RarefactFlueInFilter;
   "1DB_AIConfig".RarefactFlueOutFilter := "1DB_AIConfig_Sh".RarefactFlueOutFilter;    "Alarm_DB".RarefactFlueOutFilter := "Alarm_DB_Sh".RarefactFlueOutFilter;
   "1DB_AIConfig".PressureComprAir := "1DB_AIConfig_Sh".PressureComprAir;  "Alarm_DB".PressureComprAir := "Alarm_DB_Sh".PressureComprAir;
   "1DB_AIConfig".GasAnalyzerCO :=    "1DB_AIConfig_Sh".GasAnalyzerCO;     "Alarm_DB".GasAnalyzerCO :=    "Alarm_DB_Sh".GasAnalyzerCO;
   "1DB_AIConfig".GasAnalyzerSO2 :=   "1DB_AIConfig_Sh".GasAnalyzerSO2;    "Alarm_DB".GasAnalyzerSO2 :=   "Alarm_DB_Sh".GasAnalyzerSO2;
   "1DB_AIConfig".GasAnalyzerNOx :=   "1DB_AIConfig_Sh".GasAnalyzerNOx;    "Alarm_DB".GasAnalyzerNOx :=   "Alarm_DB_Sh".GasAnalyzerNOx;
   "1DB_AIConfig".GasAnalyzerCO2 :=   "1DB_AIConfig_Sh".GasAnalyzerCO2;    "Alarm_DB".GasAnalyzerCO2 :=   "Alarm_DB_Sh".GasAnalyzerCO2;
   "1DB_AIConfig".GasAnalyzerO2 :=    "1DB_AIConfig_Sh".GasAnalyzerO2;     "Alarm_DB".GasAnalyzerO2 :=    "Alarm_DB_Sh".GasAnalyzerO2;
   "1DB_AIConfig".FlowDustGasMix :=   "1DB_AIConfig_Sh".FlowDustGasMix;    "Alarm_DB".FlowDustGasMix :=   "Alarm_DB_Sh".FlowDustGasMix;
   "1DB_AIConfig".GasAnalyzerDust :=  "1DB_AIConfig_Sh".GasAnalyzerDust;   "Alarm_DB".GasAnalyzerDust :=  "Alarm_DB_Sh".GasAnalyzerDust;
   "1DB_AIConfig".PosValve1M :=       "1DB_AIConfig_Sh".PosValve1M;        "Alarm_DB".PosValve1M :=       "Alarm_DB_Sh".PosValve1M;
   "1DB_AIConfig".CurrentMotorShPCh1 :=    "1DB_AIConfig_Sh".CurrentMotorShPCh1;       "Alarm_DB".CurrentMotorShPCh1 :=    "Alarm_DB_Sh".CurrentMotorShPCh1;
   "1DB_AIConfig".RpmMotorShPCh1 :=   "1DB_AIConfig_Sh".RpmMotorShPCh1;    "Alarm_DB".RpmMotorShPCh1 :=   "Alarm_DB_Sh".RpmMotorShPCh1;
   "1DB_AIConfig".D1FanVibrFrontX :=  "1DB_AIConfig_Sh".D1FanVibrFrontX;   "Alarm_DB".D1FanVibrFrontX :=  "Alarm_DB_Sh".D1FanVibrFrontX;
   "1DB_AIConfig".D1FanVibrFrontY :=  "1DB_AIConfig_Sh".D1FanVibrFrontY;   "Alarm_DB".D1FanVibrFrontY :=  "Alarm_DB_Sh".D1FanVibrFrontY;
   "1DB_AIConfig".D1FanVibrBackX :=   "1DB_AIConfig_Sh".D1FanVibrBackX;    "Alarm_DB".D1FanVibrBackX :=   "Alarm_DB_Sh".D1FanVibrBackX;
   "1DB_AIConfig".D1FanVibrBackY :=   "1DB_AIConfig_Sh".D1FanVibrBackY;    "Alarm_DB".D1FanVibrBackY :=   "Alarm_DB_Sh".D1FanVibrBackY;
   "1DB_AIConfig".D1FanTempFront :=   "1DB_AIConfig_Sh".D1FanTempFront;    "Alarm_DB".D1FanTempFront :=   "Alarm_DB_Sh".D1FanTempFront;
   "1DB_AIConfig".D1FanTempBack :=    "1DB_AIConfig_Sh".D1FanTempBack;     "Alarm_DB".D1FanTempBack :=    "Alarm_DB_Sh".D1FanTempBack;
   "1DB_AIConfig".D1MotorTempFront := "1DB_AIConfig_Sh".D1MotorTempFront;  "Alarm_DB".D1MotorTempFront := "Alarm_DB_Sh".D1MotorTempFront;
   "1DB_AIConfig".D1MotorTempBack :=  "1DB_AIConfig_Sh".D1MotorTempBack;   "Alarm_DB".D1MotorTempBack :=  "Alarm_DB_Sh".D1MotorTempBack;
   "1DB_AIConfig".D1MotorTempWindA1:= "1DB_AIConfig_Sh".D1MotorTempWindA1; "Alarm_DB".D1MotorTempWindA1:= "Alarm_DB_Sh".D1MotorTempWindA1;
   "1DB_AIConfig".D1MotorTempWindA2:= "1DB_AIConfig_Sh".D1MotorTempWindA2; "Alarm_DB".D1MotorTempWindA2:= "Alarm_DB_Sh".D1MotorTempWindA2;
   "1DB_AIConfig".D1MotorTempWindB1:= "1DB_AIConfig_Sh".D1MotorTempWindB1; "Alarm_DB".D1MotorTempWindB1:= "Alarm_DB_Sh".D1MotorTempWindB1;
   "1DB_AIConfig".D1MotorTempWindB2:= "1DB_AIConfig_Sh".D1MotorTempWindB2; "Alarm_DB".D1MotorTempWindB2:= "Alarm_DB_Sh".D1MotorTempWindB2;
   "1DB_AIConfig".D1MotorTempWindC1:= "1DB_AIConfig_Sh".D1MotorTempWindC1; "Alarm_DB".D1MotorTempWindC1:= "Alarm_DB_Sh".D1MotorTempWindC1;
   "1DB_AIConfig".D1MotorTempWindC2:= "1DB_AIConfig_Sh".D1MotorTempWindC2; "Alarm_DB".D1MotorTempWindC2:= "Alarm_DB_Sh".D1MotorTempWindC2;
   "1DB_AIConfig".TGasDuctInCyclone:= "1DB_AIConfig_Sh".TGasDuctInCyclone; "Alarm_DB".TGasDuctInCyclone:= "Alarm_DB_Sh".TGasDuctInCyclone;
   "1DB_AIConfig".TGasDuctInFilter := "1DB_AIConfig_Sh".TGasDuctInFilter;  "Alarm_DB".TGasDuctInFilter := "Alarm_DB_Sh".TGasDuctInFilter;
   "1DB_AIConfig".TGasOutPipe :=      "1DB_AIConfig_Sh".TGasOutPipe;       "Alarm_DB".TGasOutPipe :=      "Alarm_DB_Sh".TGasOutPipe;

   "HMI-Machinery"."1M_PID" := "HMI-Machinery_Sh"."1M_PID";
   "HMI-Machinery".Dym_PID :=  "HMI-Machinery_Sh".Dym_PID;
END_FUNCTION

// folder: Simulation

FUNCTION "Sim1M" : Void   // FC901, LAD
{ S7_Optimized_Access := 'TRUE' }
VERSION : 0.1
   VAR_TEMP
      txOpen1M : Bool;
      txClose1M : Bool;
      txFullOpen : Bool;
      txFullClose : Bool;
   END_VAR
   VAR_TEMP   // added for the SCL form of the ladder/FBD networks
      _w1 : Bool;
      _w2 : Bool;
   END_VAR
BEGIN

REGION Network 2: Симуляция запаздывания старта МЭО на открытие
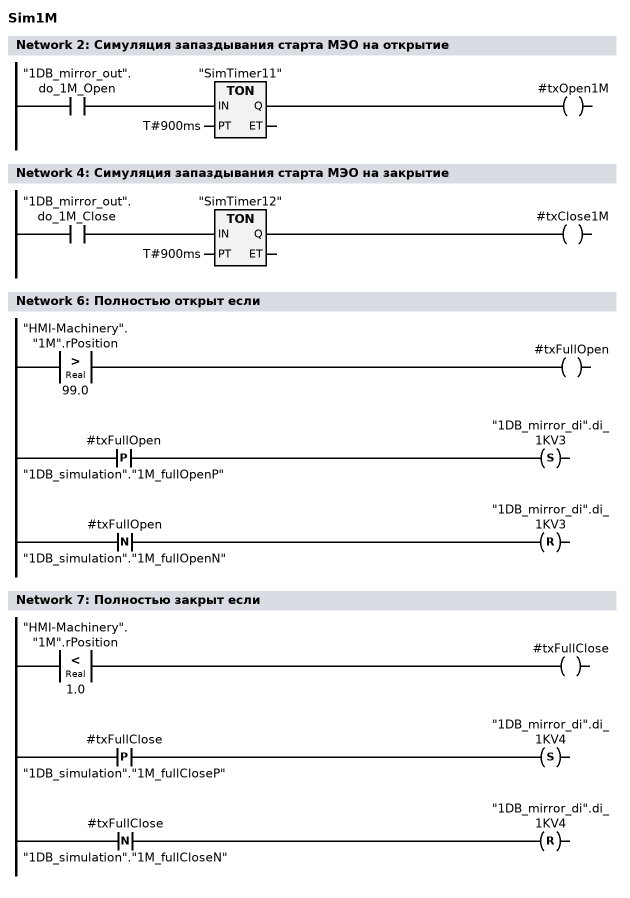
   "SimTimer11".TON(IN := "1DB_mirror_out".do_1M_Open, PT := T#900ms);
   #txOpen1M := "SimTimer11".Q;
END_REGION

REGION Network 3 (SCL): Симуляция позиции на открытие
   IF #txOpen1M AND "1DB_simulation"."1M_simPos"
                AND "iDBfor1M".ixMEO_Ready THEN
       IF "1DB_mirror_aiw".aiw_PV1M < 27648 THEN
           "1DB_mirror_aiw".aiw_PV1M += 33;
       END_IF;
   END_IF;
END_REGION

REGION Network 4: Симуляция запаздывания старта МЭО на закрытие
   "SimTimer12".TON(IN := "1DB_mirror_out".do_1M_Close, PT := T#900ms);
   #txClose1M := "SimTimer12".Q;
END_REGION

REGION Network 5 (SCL): Симуляция позиции на закрытие
   IF #txClose1M AND "1DB_simulation"."1M_simPos"
                 AND "iDBfor1M".ixMEO_Ready THEN
       IF "1DB_mirror_aiw".aiw_PV1M > 0 THEN
           "1DB_mirror_aiw".aiw_PV1M -= 33;
       END_IF;
   END_IF;
END_REGION

REGION Network 6: Полностью открыт если
   RUNG wire#powerrail
      { S7_Templates := "SrcType := Real" } GT_Contact(in1 := "HMI-Machinery"."1M".rPosition, in2 := 99.0)
      Coil( #txFullOpen )
   END_RUNG
   RUNG wire#powerrail
      P_Contact(operand := #txFullOpen, bit := "1DB_simulation"."1M_fullOpenP")
      S_Coil( "1DB_mirror_di".di_1KV3 )
   END_RUNG
   RUNG wire#powerrail
      N_Contact(operand := #txFullOpen, bit := "1DB_simulation"."1M_fullOpenN")
      R_Coil( "1DB_mirror_di".di_1KV3 )
   END_RUNG
   // the same network as SCL:
   #txFullOpen := "HMI-Machinery"."1M".rPosition > 99.0;
   #_w1 := #txFullOpen AND NOT "1DB_simulation"."1M_fullOpenP";   // rising edge of #txFullOpen
   "1DB_simulation"."1M_fullOpenP" := #txFullOpen;
   IF #_w1 THEN "1DB_mirror_di".di_1KV3 := TRUE; END_IF;
   #_w2 := NOT #txFullOpen AND "1DB_simulation"."1M_fullOpenN";   // falling edge of #txFullOpen
   "1DB_simulation"."1M_fullOpenN" := #txFullOpen;
   IF #_w2 THEN "1DB_mirror_di".di_1KV3 := FALSE; END_IF;
END_REGION

REGION Network 7: Полностью закрыт если
   RUNG wire#powerrail
      { S7_Templates := "SrcType := Real" } LT_Contact(in1 := "HMI-Machinery"."1M".rPosition, in2 := 1.0)
      Coil( #txFullClose )
   END_RUNG
   RUNG wire#powerrail
      P_Contact(operand := #txFullClose, bit := "1DB_simulation"."1M_fullCloseP")
      S_Coil( "1DB_mirror_di".di_1KV4 )
   END_RUNG
   RUNG wire#powerrail
      N_Contact(operand := #txFullClose, bit := "1DB_simulation"."1M_fullCloseN")
      R_Coil( "1DB_mirror_di".di_1KV4 )
   END_RUNG
   // the same network as SCL:
   #txFullClose := "HMI-Machinery"."1M".rPosition < 1.0;
   #_w1 := #txFullClose AND NOT "1DB_simulation"."1M_fullCloseP";   // rising edge of #txFullClose
   "1DB_simulation"."1M_fullCloseP" := #txFullClose;
   IF #_w1 THEN "1DB_mirror_di".di_1KV4 := TRUE; END_IF;
   #_w2 := NOT #txFullClose AND "1DB_simulation"."1M_fullCloseN";   // falling edge of #txFullClose
   "1DB_simulation"."1M_fullCloseN" := #txFullClose;
   IF #_w2 THEN "1DB_mirror_di".di_1KV4 := FALSE; END_IF;
END_REGION

REGION Network 9 (SCL): Симуляция температуры перед фильтром
   IF "HMI-Machinery"."1M".rPosition >45.0 AND "1DB_mirror_aiw".aiw_TE102a >1000
       AND "1DB_simulation"."1M_simTE102" THEN
       "1DB_mirror_aiw".aiw_TE102a -= 1;
   ELSIF "HMI-Machinery"."1M".rPosition <45.0 AND "1DB_mirror_aiw".aiw_TE102a <2800
       AND "1DB_simulation"."1M_simTE102" THEN
       "1DB_mirror_aiw".aiw_TE102a += 1;
   END_IF;
END_REGION
END_FUNCTION

FUNCTION "Sim2M" : Void   // FC902, LAD
{ S7_Optimized_Access := 'TRUE' }
VERSION : 0.1
   VAR_TEMP   // added for the SCL form of the ladder/FBD networks
      _w1 : Bool;
   END_VAR
BEGIN

REGION Network 2: Симуляция открытия
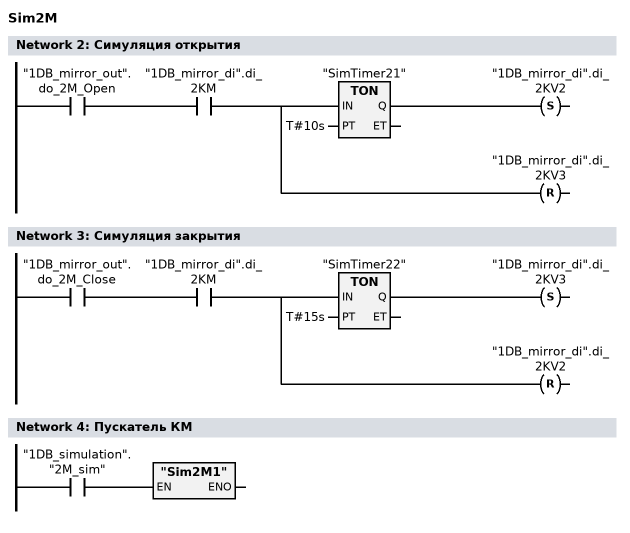
   #_w1 := "1DB_mirror_out".do_2M_Open AND "1DB_mirror_di".di_2KM;
   "SimTimer21".TON(IN := #_w1, PT := T#10s);
   IF "SimTimer21".Q THEN "1DB_mirror_di".di_2KV2 := TRUE; END_IF;
   IF #_w1 THEN "1DB_mirror_di".di_2KV3 := FALSE; END_IF;
END_REGION

REGION Network 3: Симуляция закрытия
   #_w1 := "1DB_mirror_out".do_2M_Close AND "1DB_mirror_di".di_2KM;
   "SimTimer22".TON(IN := #_w1, PT := T#15s);
   IF "SimTimer22".Q THEN "1DB_mirror_di".di_2KV3 := TRUE; END_IF;
   IF #_w1 THEN "1DB_mirror_di".di_2KV2 := FALSE; END_IF;
END_REGION

REGION Network 4: Пускатель КМ
   RUNG wire#powerrail
      Contact( "1DB_simulation"."2M_sim" )
      "Sim2M1"()
   END_RUNG
   // the same network as SCL:
   IF "1DB_simulation"."2M_sim" THEN "Sim2M1"(); END_IF;
END_REGION
END_FUNCTION

FUNCTION "Sim3-8M" : Void   // FC903, LAD
{ S7_Optimized_Access := 'TRUE' }
VERSION : 0.1
BEGIN

REGION Network 2: Пускатели
